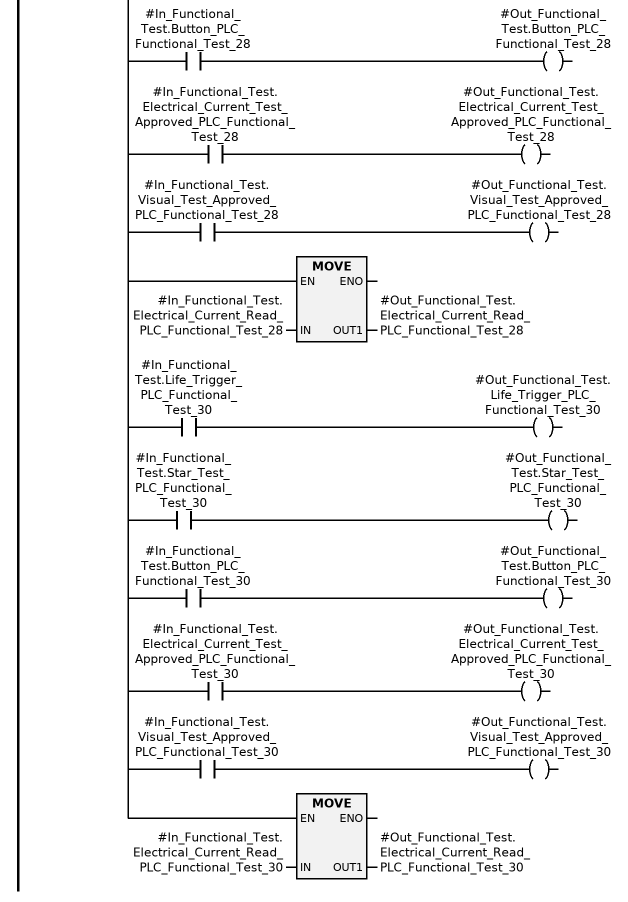
   RUNG wire#powerrail
      { S7_Templates := "SrcType := SInt" } EQ_Contact(in1 := #Test_Station, in2 := 14)
      wire#w1
      Contact( #Life_Trigger )
      Coil( #Out_Functional_Test.Life_Trigger_PLC_Functional_Test_14 )
   END_RUNG
   RUNG wire#w1
      Contact( #Star_Test )
      Coil( #Out_Functional_Test.Star_Test_PLC_Functional_Test_14 )
   END_RUNG
   RUNG wire#w1
      Contact( #Button_Start_Approve )
      Coil( #Out_Functional_Test.Button_PLC_Functional_Test_14 )
   END_RUNG
   RUNG wire#w1
      Contact( #Electrical_Current_Test_Approved )
      Coil( #Out_Functional_Test.Electrical_Current_Test_Approved_PLC_Functional_Test_14 )
   END_RUNG
   RUNG wire#w1
      Contact( #Visual_Test_Approved )
      Coil( #Out_Functional_Test.Visual_Test_Approved_PLC_Functional_Test_14 )
   END_RUNG
   RUNG wire#w1
      Contact( #In_Test_Parameters.Reset_PLC_Functional_Test_14 )
      Coil( #Reset_Functional_Test )
   END_RUNG
   RUNG wire#w1
      Move(in := #Electrical_Current_Read, out1 => #Out_Functional_Test.Electrical_Current_Read_PLC_Functional_Test_14)
   END_RUNG
   RUNG wire#w1
      Contact( #In_Functional_Test.Life_Trigger_PLC_Functional_Test_16 )
      Coil( #Out_Functional_Test.Life_Trigger_PLC_Functional_Test_16 )
   END_RUNG
   RUNG wire#w1
      Contact( #In_Functional_Test.Star_Test_PLC_Functional_Test_16 )
      Coil( #Out_Functional_Test.Star_Test_PLC_Functional_Test_16 )
   END_RUNG
   RUNG wire#w1
      Contact( #In_Functional_Test.Button_PLC_Functional_Test_16 )
      Coil( #Out_Functional_Test.Button_PLC_Functional_Test_16 )
   END_RUNG
   RUNG wire#w1
      Contact( #In_Functional_Test.Electrical_Current_Test_Approved_PLC_Functional_Test_16 )
      Coil( #Out_Functional_Test.Electrical_Current_Test_Approved_PLC_Functional_Test_16 )
   END_RUNG
   RUNG wire#w1
      Contact( #In_Functional_Test.Visual_Test_Approved_PLC_Functional_Test_16 )
      Coil( #Out_Functional_Test.Visual_Test_Approved_PLC_Functional_Test_16 )
   END_RUNG
   RUNG wire#w1
      Move(in := #In_Functional_Test.Electrical_Current_Read_PLC_Functional_Test_16, out1 => #Out_Functional_Test.Electrical_Current_Read_PLC_Functional_Test_16)
   END_RUNG
   RUNG wire#w1
      Contact( #In_Functional_Test.Life_Trigger_PLC_Functional_Test_18 )
      Coil( #Out_Functional_Test.Life_Trigger_PLC_Functional_Test_18 )
   END_RUNG
   RUNG wire#w1
      Contact( #In_Functional_Test.Star_Test_PLC_Functional_Test_18 )
      Coil( #Out_Functional_Test.Star_Test_PLC_Functional_Test_18 )
   END_RUNG
   RUNG wire#w1
      Contact( #In_Functional_Test.Button_PLC_Functional_Test_18 )
      Coil( #Out_Functional_Test.Button_PLC_Functional_Test_18 )
   END_RUNG
   RUNG wire#w1
      Contact( #In_Functional_Test.Electrical_Current_Test_Approved_PLC_Functional_Test_18 )
      Coil( #Out_Functional_Test.Electrical_Current_Test_Approved_PLC_Functional_Test_18 )
   END_RUNG
   RUNG wire#w1
      Contact( #In_Functional_Test.Visual_Test_Approved_PLC_Functional_Test_18 )
      Coil( #Out_Functional_Test.Visual_Test_Approved_PLC_Functional_Test_18 )
   END_RUNG
   RUNG wire#w1
      Move(in := #In_Functional_Test.Electrical_Current_Read_PLC_Functional_Test_18, out1 => #Out_Functional_Test.Electrical_Current_Read_PLC_Functional_Test_18)
   END_RUNG
   RUNG wire#w1
      Contact( #In_Functional_Test.Life_Trigger_PLC_Functional_Test_20 )
      Coil( #Out_Functional_Test.Life_Trigger_PLC_Functional_Test_20 )
   END_RUNG
   RUNG wire#w1
      Contact( #In_Functional_Test.Star_Test_PLC_Functional_Test_20 )
      Coil( #Out_Functional_Test.Star_Test_PLC_Functional_Test_20 )
   END_RUNG
   RUNG wire#w1
      Contact( #In_Functional_Test.Button_PLC_Functional_Test_20 )
      Coil( #Out_Functional_Test.Button_PLC_Functional_Test_20 )
   END_RUNG
   RUNG wire#w1
      Contact( #In_Functional_Test.Electrical_Current_Test_Approved_PLC_Functional_Test_20 )
      Coil( #Out_Functional_Test.Electrical_Current_Test_Approved_PLC_Functional_Test_20 )
   END_RUNG
   RUNG wire#w1
      Contact( #In_Functional_Test.Visual_Test_Approved_PLC_Functional_Test_20 )
      Coil( #Out_Functional_Test.Visual_Test_Approved_PLC_Functional_Test_20 )
   END_RUNG
   RUNG wire#w1
      Move(in := #In_Functional_Test.Electrical_Current_Read_PLC_Functional_Test_20, out1 => #Out_Functional_Test.Electrical_Current_Read_PLC_Functional_Test_20)
   END_RUNG
   RUNG wire#w1
      Contact( #In_Functional_Test.Life_Trigger_PLC_Functional_Test_22 )
      Coil( #Out_Functional_Test.Life_Trigger_PLC_Functional_Test_22 )
   END_RUNG
   RUNG wire#w1
      Contact( #In_Functional_Test.Star_Test_PLC_Functional_Test_22 )
      Coil( #Out_Functional_Test.Star_Test_PLC_Functional_Test_22 )
   END_RUNG
   RUNG wire#w1
      Contact( #In_Functional_Test.Button_PLC_Functional_Test_22 )
      Coil( #Out_Functional_Test.Button_PLC_Functional_Test_22 )
   END_RUNG
   RUNG wire#w1
      Contact( #In_Functional_Test.Electrical_Current_Test_Approved_PLC_Functional_Test_22 )
      Coil( #Out_Functional_Test.Electrical_Current_Test_Approved_PLC_Functional_Test_22 )
   END_RUNG
   RUNG wire#w1
      Contact( #In_Functional_Test.Visual_Test_Approved_PLC_Functional_Test_22 )
      Coil( #Out_Functional_Test.Visual_Test_Approved_PLC_Functional_Test_22 )
   END_RUNG
   RUNG wire#w1
      Move(in := #In_Functional_Test.Electrical_Current_Read_PLC_Functional_Test_22, out1 => #Out_Functional_Test.Electrical_Current_Read_PLC_Functional_Test_22)
   END_RUNG
   RUNG wire#w1
      Contact( #In_Functional_Test.Life_Trigger_PLC_Functional_Test_24 )
      Coil( #Out_Functional_Test.Life_Trigger_PLC_Functional_Test_24 )
   END_RUNG
   RUNG wire#w1
      Contact( #In_Functional_Test.Star_Test_PLC_Functional_Test_24 )
      Coil( #Out_Functional_Test.Star_Test_PLC_Functional_Test_24 )
   END_RUNG
   RUNG wire#w1
      Contact( #In_Functional_Test.Button_PLC_Functional_Test_24 )
      Coil( #Out_Functional_Test.Button_PLC_Functional_Test_24 )
   END_RUNG
   RUNG wire#w1
      Contact( #In_Functional_Test.Electrical_Current_Test_Approved_PLC_Functional_Test_24 )
      Coil( #Out_Functional_Test.Electrical_Current_Test_Approved_PLC_Functional_Test_24 )
   END_RUNG
   RUNG wire#w1
      Contact( #In_Functional_Test.Visual_Test_Approved_PLC_Functional_Test_24 )
      Coil( #Out_Functional_Test.Visual_Test_Approved_PLC_Functional_Test_24 )
   END_RUNG
   RUNG wire#w1
      Move(in := #In_Functional_Test.Electrical_Current_Read_PLC_Functional_Test_24, out1 => #Out_Functional_Test.Electrical_Current_Read_PLC_Functional_Test_24)
   END_RUNG
   RUNG wire#w1
      Contact( #In_Functional_Test.Life_Trigger_PLC_Functional_Test_26 )
      Coil( #Out_Functional_Test.Life_Trigger_PLC_Functional_Test_26 )
   END_RUNG
   RUNG wire#w1
      Contact( #In_Functional_Test.Star_Test_PLC_Functional_Test_26 )
      Coil( #Out_Functional_Test.Star_Test_PLC_Functional_Test_26 )
   END_RUNG
   RUNG wire#w1
      Contact( #In_Functional_Test.Button_PLC_Functional_Test_26 )
      Coil( #Out_Functional_Test.Button_PLC_Functional_Test_26 )
   END_RUNG
   RUNG wire#w1
      Contact( #In_Functional_Test.Electrical_Current_Test_Approved_PLC_Functional_Test_26 )
      Coil( #Out_Functional_Test.Electrical_Current_Test_Approved_PLC_Functional_Test_26 )
   END_RUNG
   RUNG wire#w1
      Contact( #In_Functional_Test.Visual_Test_Approved_PLC_Functional_Test_26 )
      Coil( #Out_Functional_Test.Visual_Test_Approved_PLC_Functional_Test_26 )
   END_RUNG
   RUNG wire#w1
      Move(in := #In_Functional_Test.Electrical_Current_Read_PLC_Functional_Test_26, out1 => #Out_Functional_Test.Electrical_Current_Read_PLC_Functional_Test_26)
   END_RUNG
   RUNG wire#w1
      Contact( #In_Functional_Test.Life_Trigger_PLC_Functional_Test_28 )
      Coil( #Out_Functional_Test.Life_Trigger_PLC_Functional_Test_28 )
   END_RUNG
   RUNG wire#w1
      Contact( #In_Functional_Test.Star_Test_PLC_Functional_Test_28 )
      Coil( #Out_Functional_Test.Star_Test_PLC_Functional_Test_28 )
   END_RUNG
   RUNG wire#w1
      Contact( #In_Functional_Test.Button_PLC_Functional_Test_28 )
      Coil( #Out_Functional_Test.Button_PLC_Functional_Test_28 )
   END_RUNG
   RUNG wire#w1
      Contact( #In_Functional_Test.Electrical_Current_Test_Approved_PLC_Functional_Test_28 )
      Coil( #Out_Functional_Test.Electrical_Current_Test_Approved_PLC_Functional_Test_28 )
   END_RUNG
   RUNG wire#w1
      Contact( #In_Functional_Test.Visual_Test_Approved_PLC_Functional_Test_28 )
      Coil( #Out_Functional_Test.Visual_Test_Approved_PLC_Functional_Test_28 )
   END_RUNG
   RUNG wire#w1
      Move(in := #In_Functional_Test.Electrical_Current_Read_PLC_Functional_Test_28, out1 => #Out_Functional_Test.Electrical_Current_Read_PLC_Functional_Test_28)
   END_RUNG
   RUNG wire#w1
      Contact( #In_Functional_Test.Life_Trigger_PLC_Functional_Test_30 )
      Coil( #Out_Functional_Test.Life_Trigger_PLC_Functional_Test_30 )
   END_RUNG
   RUNG wire#w1
      Contact( #In_Functional_Test.Star_Test_PLC_Functional_Test_30 )
      Coil( #Out_Functional_Test.Star_Test_PLC_Functional_Test_30 )
   END_RUNG
   RUNG wire#w1
      Contact( #In_Functional_Test.Button_PLC_Functional_Test_30 )
      Coil( #Out_Functional_Test.Button_PLC_Functional_Test_30 )
   END_RUNG
   RUNG wire#w1
      Contact( #In_Functional_Test.Electrical_Current_Test_Approved_PLC_Functional_Test_30 )
      Coil( #Out_Functional_Test.Electrical_Current_Test_Approved_PLC_Functional_Test_30 )
   END_RUNG
   RUNG wire#w1
      Contact( #In_Functional_Test.Visual_Test_Approved_PLC_Functional_Test_30 )
      Coil( #Out_Functional_Test.Visual_Test_Approved_PLC_Functional_Test_30 )
   END_RUNG
   RUNG wire#w1
      Move(in := #In_Functional_Test.Electrical_Current_Read_PLC_Functional_Test_30, out1 => #Out_Functional_Test.Electrical_Current_Read_PLC_Functional_Test_30)
   END_RUNG
   // the same network as SCL:
   #_w1 := #Test_Station = 14;
   #Out_Functional_Test.Life_Trigger_PLC_Functional_Test_14 := #_w1 AND #Life_Trigger;
   #Out_Functional_Test.Star_Test_PLC_Functional_Test_14 := #_w1 AND #Star_Test;
   #Out_Functional_Test.Button_PLC_Functional_Test_14 := #_w1 AND #Button_Start_Approve;
   #Out_Functional_Test.Electrical_Current_Test_Approved_PLC_Functional_Test_14 := #_w1 AND #Electrical_Current_Test_Approved;
   #Out_Functional_Test.Visual_Test_Approved_PLC_Functional_Test_14 := #_w1 AND #Visual_Test_Approved;
   #Reset_Functional_Test := #_w1 AND #In_Test_Parameters.Reset_PLC_Functional_Test_14;
   IF #_w1 THEN
       #Out_Functional_Test.Electrical_Current_Read_PLC_Functional_Test_14 := #Electrical_Current_Read;
   END_IF;
   #Out_Functional_Test.Life_Trigger_PLC_Functional_Test_16 := #_w1 AND #In_Functional_Test.Life_Trigger_PLC_Functional_Test_16;
   #Out_Functional_Test.Star_Test_PLC_Functional_Test_16 := #_w1 AND #In_Functional_Test.Star_Test_PLC_Functional_Test_16;
   #Out_Functional_Test.Button_PLC_Functional_Test_16 := #_w1 AND #In_Functional_Test.Button_PLC_Functional_Test_16;
   #Out_Functional_Test.Electrical_Current_Test_Approved_PLC_Functional_Test_16 := #_w1 AND #In_Functional_Test.Electrical_Current_Test_Approved_PLC_Functional_Test_16;
   #Out_Functional_Test.Visual_Test_Approved_PLC_Functional_Test_16 := #_w1 AND #In_Functional_Test.Visual_Test_Approved_PLC_Functional_Test_16;
   IF #_w1 THEN
       #Out_Functional_Test.Electrical_Current_Read_PLC_Functional_Test_16 := #In_Functional_Test.Electrical_Current_Read_PLC_Functional_Test_16;
   END_IF;
   #Out_Functional_Test.Life_Trigger_PLC_Functional_Test_18 := #_w1 AND #In_Functional_Test.Life_Trigger_PLC_Functional_Test_18;
   #Out_Functional_Test.Star_Test_PLC_Functional_Test_18 := #_w1 AND #In_Functional_Test.Star_Test_PLC_Functional_Test_18;
   #Out_Functional_Test.Button_PLC_Functional_Test_18 := #_w1 AND #In_Functional_Test.Button_PLC_Functional_Test_18;
   #Out_Functional_Test.Electrical_Current_Test_Approved_PLC_Functional_Test_18 := #_w1 AND #In_Functional_Test.Electrical_Current_Test_Approved_PLC_Functional_Test_18;
   #Out_Functional_Test.Visual_Test_Approved_PLC_Functional_Test_18 := #_w1 AND #In_Functional_Test.Visual_Test_Approved_PLC_Functional_Test_18;
   IF #_w1 THEN
       #Out_Functional_Test.Electrical_Current_Read_PLC_Functional_Test_18 := #In_Functional_Test.Electrical_Current_Read_PLC_Functional_Test_18;
   END_IF;
   #Out_Functional_Test.Life_Trigger_PLC_Functional_Test_20 := #_w1 AND #In_Functional_Test.Life_Trigger_PLC_Functional_Test_20;
   #Out_Functional_Test.Star_Test_PLC_Functional_Test_20 := #_w1 AND #In_Functional_Test.Star_Test_PLC_Functional_Test_20;
   #Out_Functional_Test.Button_PLC_Functional_Test_20 := #_w1 AND #In_Functional_Test.Button_PLC_Functional_Test_20;
   #Out_Functional_Test.Electrical_Current_Test_Approved_PLC_Functional_Test_20 := #_w1 AND #In_Functional_Test.Electrical_Current_Test_Approved_PLC_Functional_Test_20;
   #Out_Functional_Test.Visual_Test_Approved_PLC_Functional_Test_20 := #_w1 AND #In_Functional_Test.Visual_Test_Approved_PLC_Functional_Test_20;
   IF #_w1 THEN
       #Out_Functional_Test.Electrical_Current_Read_PLC_Functional_Test_20 := #In_Functional_Test.Electrical_Current_Read_PLC_Functional_Test_20;
   END_IF;
   #Out_Functional_Test.Life_Trigger_PLC_Functional_Test_22 := #_w1 AND #In_Functional_Test.Life_Trigger_PLC_Functional_Test_22;
   #Out_Functional_Test.Star_Test_PLC_Functional_Test_22 := #_w1 AND #In_Functional_Test.Star_Test_PLC_Functional_Test_22;
   #Out_Functional_Test.Button_PLC_Functional_Test_22 := #_w1 AND #In_Functional_Test.Button_PLC_Functional_Test_22;
   #Out_Functional_Test.Electrical_Current_Test_Approved_PLC_Functional_Test_22 := #_w1 AND #In_Functional_Test.Electrical_Current_Test_Approved_PLC_Functional_Test_22;
   #Out_Functional_Test.Visual_Test_Approved_PLC_Functional_Test_22 := #_w1 AND #In_Functional_Test.Visual_Test_Approved_PLC_Functional_Test_22;
   IF #_w1 THEN
       #Out_Functional_Test.Electrical_Current_Read_PLC_Functional_Test_22 := #In_Functional_Test.Electrical_Current_Read_PLC_Functional_Test_22;
   END_IF;
   #Out_Functional_Test.Life_Trigger_PLC_Functional_Test_24 := #_w1 AND #In_Functional_Test.Life_Trigger_PLC_Functional_Test_24;
   #Out_Functional_Test.Star_Test_PLC_Functional_Test_24 := #_w1 AND #In_Functional_Test.Star_Test_PLC_Functional_Test_24;
   #Out_Functional_Test.Button_PLC_Functional_Test_24 := #_w1 AND #In_Functional_Test.Button_PLC_Functional_Test_24;
   #Out_Functional_Test.Electrical_Current_Test_Approved_PLC_Functional_Test_24 := #_w1 AND #In_Functional_Test.Electrical_Current_Test_Approved_PLC_Functional_Test_24;
   #Out_Functional_Test.Visual_Test_Approved_PLC_Functional_Test_24 := #_w1 AND #In_Functional_Test.Visual_Test_Approved_PLC_Functional_Test_24;
   IF #_w1 THEN
       #Out_Functional_Test.Electrical_Current_Read_PLC_Functional_Test_24 := #In_Functional_Test.Electrical_Current_Read_PLC_Functional_Test_24;
   END_IF;
   #Out_Functional_Test.Life_Trigger_PLC_Functional_Test_26 := #_w1 AND #In_Functional_Test.Life_Trigger_PLC_Functional_Test_26;
   #Out_Functional_Test.Star_Test_PLC_Functional_Test_26 := #_w1 AND #In_Functional_Test.Star_Test_PLC_Functional_Test_26;
   #Out_Functional_Test.Button_PLC_Functional_Test_26 := #_w1 AND #In_Functional_Test.Button_PLC_Functional_Test_26;
   #Out_Functional_Test.Electrical_Current_Test_Approved_PLC_Functional_Test_26 := #_w1 AND #In_Functional_Test.Electrical_Current_Test_Approved_PLC_Functional_Test_26;
   #Out_Functional_Test.Visual_Test_Approved_PLC_Functional_Test_26 := #_w1 AND #In_Functional_Test.Visual_Test_Approved_PLC_Functional_Test_26;
   IF #_w1 THEN
       #Out_Functional_Test.Electrical_Current_Read_PLC_Functional_Test_26 := #In_Functional_Test.Electrical_Current_Read_PLC_Functional_Test_26;
   END_IF;
   #Out_Functional_Test.Life_Trigger_PLC_Functional_Test_28 := #_w1 AND #In_Functional_Test.Life_Trigger_PLC_Functional_Test_28;
   #Out_Functional_Test.Star_Test_PLC_Functional_Test_28 := #_w1 AND #In_Functional_Test.Star_Test_PLC_Functional_Test_28;
   #Out_Functional_Test.Button_PLC_Functional_Test_28 := #_w1 AND #In_Functional_Test.Button_PLC_Functional_Test_28;
   #Out_Functional_Test.Electrical_Current_Test_Approved_PLC_Functional_Test_28 := #_w1 AND #In_Functional_Test.Electrical_Current_Test_Approved_PLC_Functional_Test_28;
   #Out_Functional_Test.Visual_Test_Approved_PLC_Functional_Test_28 := #_w1 AND #In_Functional_Test.Visual_Test_Approved_PLC_Functional_Test_28;
   IF #_w1 THEN
       #Out_Functional_Test.Electrical_Current_Read_PLC_Functional_Test_28 := #In_Functional_Test.Electrical_Current_Read_PLC_Functional_Test_28;
   END_IF;
   #Out_Functional_Test.Life_Trigger_PLC_Functional_Test_30 := #_w1 AND #In_Functional_Test.Life_Trigger_PLC_Functional_Test_30;
   #Out_Functional_Test.Star_Test_PLC_Functional_Test_30 := #_w1 AND #In_Functional_Test.Star_Test_PLC_Functional_Test_30;
   #Out_Functional_Test.Button_PLC_Functional_Test_30 := #_w1 AND #In_Functional_Test.Button_PLC_Functional_Test_30;
   #Out_Functional_Test.Electrical_Current_Test_Approved_PLC_Functional_Test_30 := #_w1 AND #In_Functional_Test.Electrical_Current_Test_Approved_PLC_Functional_Test_30;
   #Out_Functional_Test.Visual_Test_Approved_PLC_Functional_Test_30 := #_w1 AND #In_Functional_Test.Visual_Test_Approved_PLC_Functional_Test_30;
   IF #_w1 THEN
       #Out_Functional_Test.Electrical_Current_Read_PLC_Functional_Test_30 := #In_Functional_Test.Electrical_Current_Read_PLC_Functional_Test_30;
   END_IF;
END_REGION

REGION Network 9: Functional Test Station 16
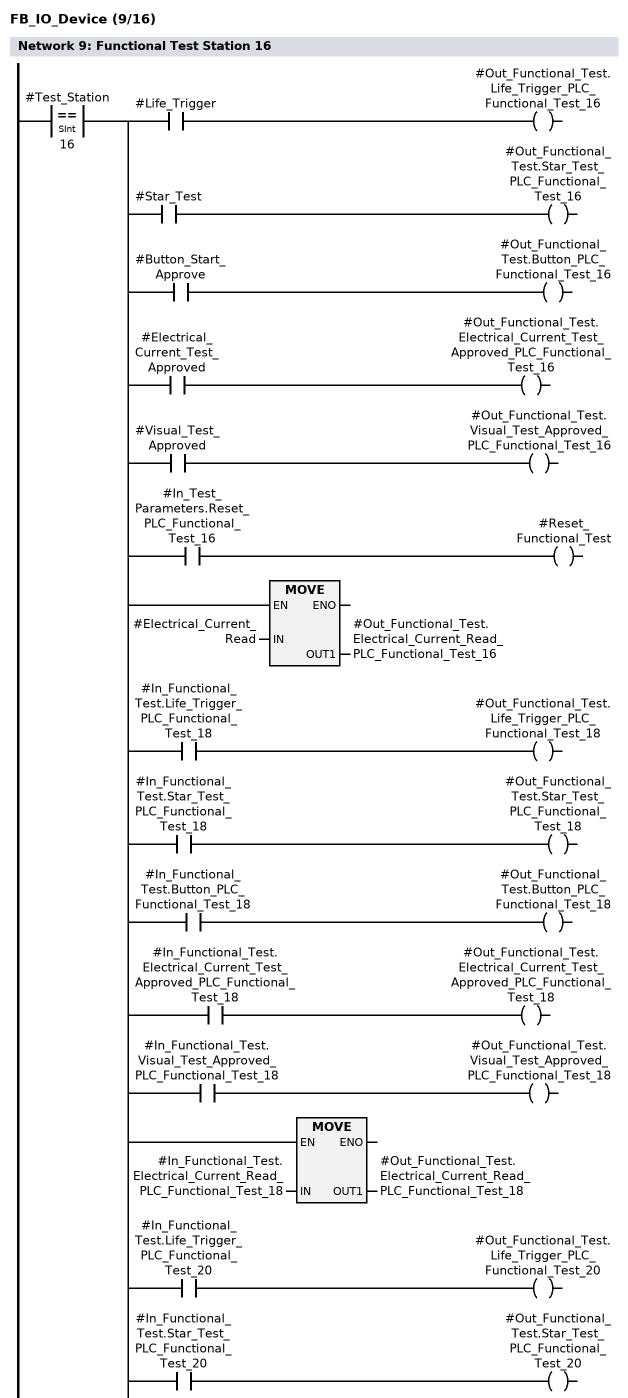
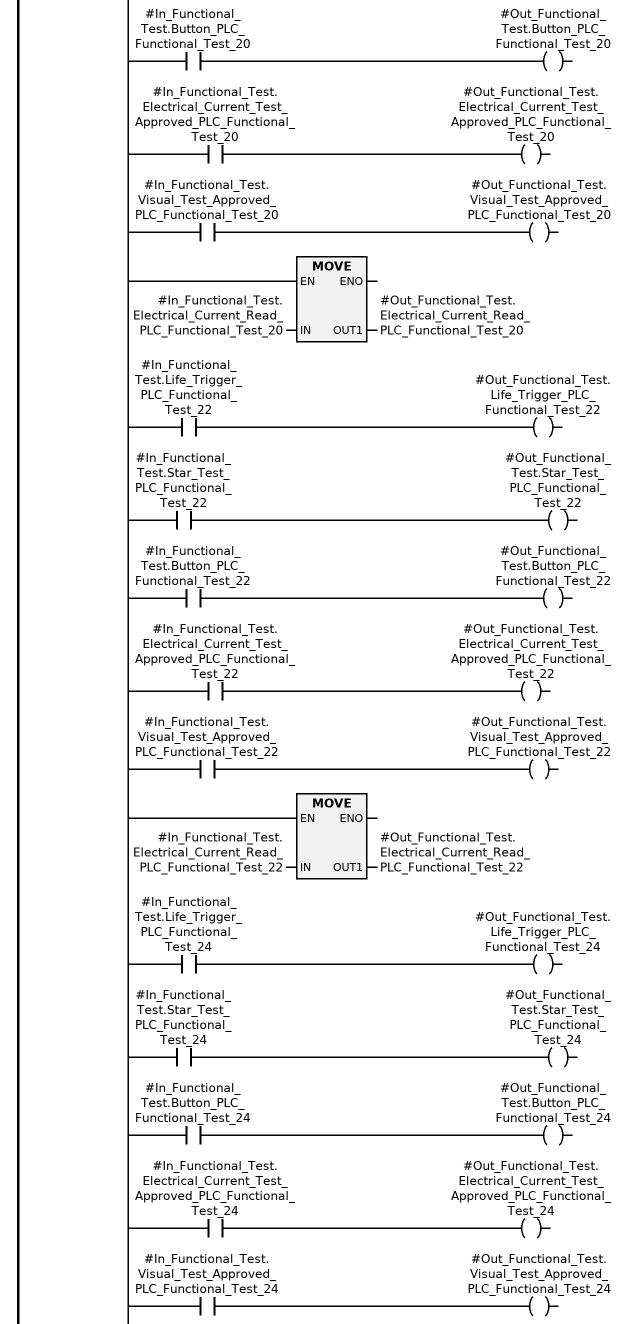
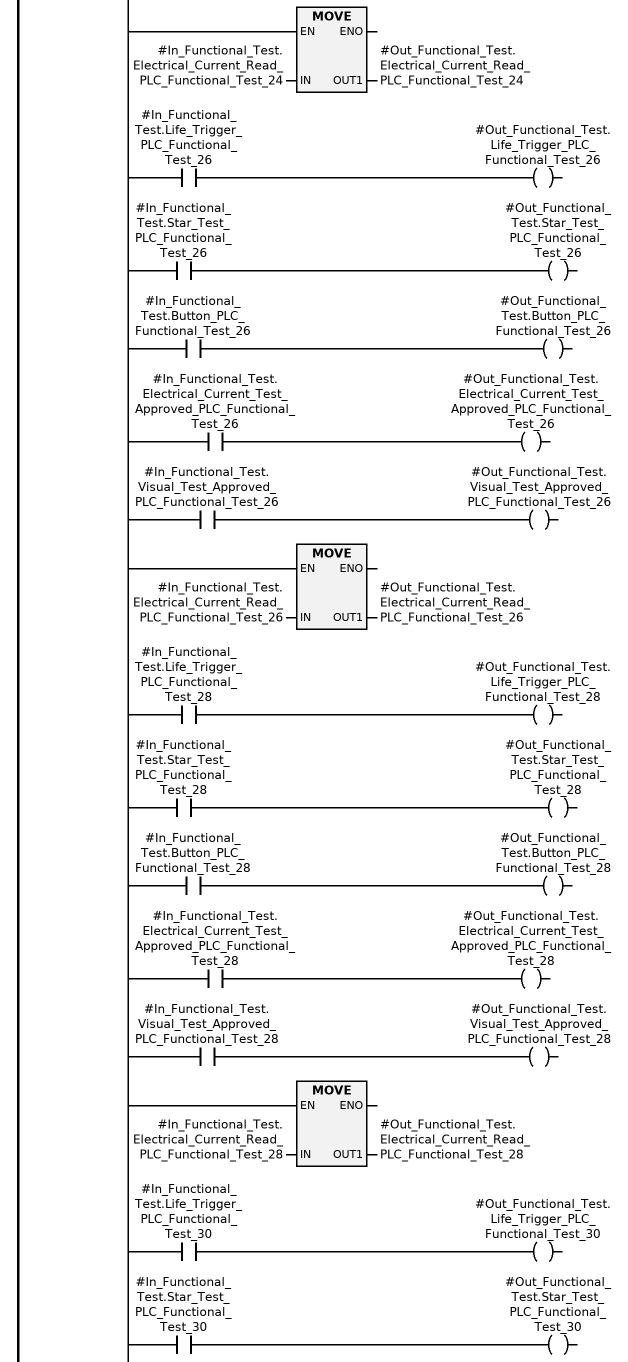
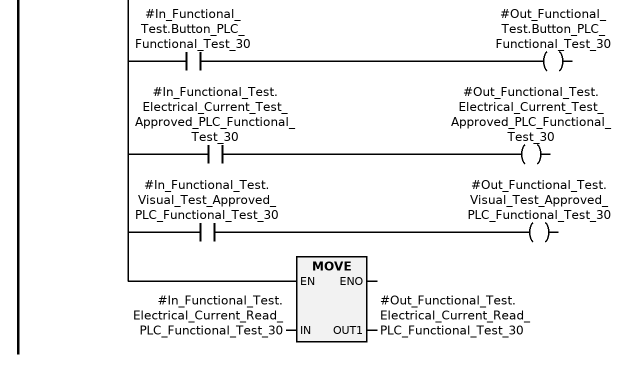
   RUNG wire#powerrail
      { S7_Templates := "SrcType := SInt" } EQ_Contact(in1 := #Test_Station, in2 := 16)
      wire#w1
      Contact( #Life_Trigger )
      Coil( #Out_Functional_Test.Life_Trigger_PLC_Functional_Test_16 )
   END_RUNG
   RUNG wire#w1
      Contact( #Star_Test )
      Coil( #Out_Functional_Test.Star_Test_PLC_Functional_Test_16 )
   END_RUNG
   RUNG wire#w1
      Contact( #Button_Start_Approve )
      Coil( #Out_Functional_Test.Button_PLC_Functional_Test_16 )
   END_RUNG
   RUNG wire#w1
      Contact( #Electrical_Current_Test_Approved )
      Coil( #Out_Functional_Test.Electrical_Current_Test_Approved_PLC_Functional_Test_16 )
   END_RUNG
   RUNG wire#w1
      Contact( #Visual_Test_Approved )
      Coil( #Out_Functional_Test.Visual_Test_Approved_PLC_Functional_Test_16 )
   END_RUNG
   RUNG wire#w1
      Contact( #In_Test_Parameters.Reset_PLC_Functional_Test_16 )
      Coil( #Reset_Functional_Test )
   END_RUNG
   RUNG wire#w1
      Move(in := #Electrical_Current_Read, out1 => #Out_Functional_Test.Electrical_Current_Read_PLC_Functional_Test_16)
   END_RUNG
   RUNG wire#w1
      Contact( #In_Functional_Test.Life_Trigger_PLC_Functional_Test_18 )
      Coil( #Out_Functional_Test.Life_Trigger_PLC_Functional_Test_18 )
   END_RUNG
   RUNG wire#w1
      Contact( #In_Functional_Test.Star_Test_PLC_Functional_Test_18 )
      Coil( #Out_Functional_Test.Star_Test_PLC_Functional_Test_18 )
   END_RUNG
   RUNG wire#w1
      Contact( #In_Functional_Test.Button_PLC_Functional_Test_18 )
      Coil( #Out_Functional_Test.Button_PLC_Functional_Test_18 )
   END_RUNG
   RUNG wire#w1
      Contact( #In_Functional_Test.Electrical_Current_Test_Approved_PLC_Functional_Test_18 )
      Coil( #Out_Functional_Test.Electrical_Current_Test_Approved_PLC_Functional_Test_18 )
   END_RUNG
   RUNG wire#w1
      Contact( #In_Functional_Test.Visual_Test_Approved_PLC_Functional_Test_18 )
      Coil( #Out_Functional_Test.Visual_Test_Approved_PLC_Functional_Test_18 )
   END_RUNG
   RUNG wire#w1
      Move(in := #In_Functional_Test.Electrical_Current_Read_PLC_Functional_Test_18, out1 => #Out_Functional_Test.Electrical_Current_Read_PLC_Functional_Test_18)
   END_RUNG
   RUNG wire#w1
      Contact( #In_Functional_Test.Life_Trigger_PLC_Functional_Test_20 )
      Coil( #Out_Functional_Test.Life_Trigger_PLC_Functional_Test_20 )
   END_RUNG
   RUNG wire#w1
      Contact( #In_Functional_Test.Star_Test_PLC_Functional_Test_20 )
      Coil( #Out_Functional_Test.Star_Test_PLC_Functional_Test_20 )
   END_RUNG
   RUNG wire#w1
      Contact( #In_Functional_Test.Button_PLC_Functional_Test_20 )
      Coil( #Out_Functional_Test.Button_PLC_Functional_Test_20 )
   END_RUNG
   RUNG wire#w1
      Contact( #In_Functional_Test.Electrical_Current_Test_Approved_PLC_Functional_Test_20 )
      Coil( #Out_Functional_Test.Electrical_Current_Test_Approved_PLC_Functional_Test_20 )
   END_RUNG
   RUNG wire#w1
      Contact( #In_Functional_Test.Visual_Test_Approved_PLC_Functional_Test_20 )
      Coil( #Out_Functional_Test.Visual_Test_Approved_PLC_Functional_Test_20 )
   END_RUNG
   RUNG wire#w1
      Move(in := #In_Functional_Test.Electrical_Current_Read_PLC_Functional_Test_20, out1 => #Out_Functional_Test.Electrical_Current_Read_PLC_Functional_Test_20)
   END_RUNG
   RUNG wire#w1
      Contact( #In_Functional_Test.Life_Trigger_PLC_Functional_Test_22 )
      Coil( #Out_Functional_Test.Life_Trigger_PLC_Functional_Test_22 )
   END_RUNG
   RUNG wire#w1
      Contact( #In_Functional_Test.Star_Test_PLC_Functional_Test_22 )
      Coil( #Out_Functional_Test.Star_Test_PLC_Functional_Test_22 )
   END_RUNG
   RUNG wire#w1
      Contact( #In_Functional_Test.Button_PLC_Functional_Test_22 )
      Coil( #Out_Functional_Test.Button_PLC_Functional_Test_22 )
   END_RUNG
   RUNG wire#w1
      Contact( #In_Functional_Test.Electrical_Current_Test_Approved_PLC_Functional_Test_22 )
      Coil( #Out_Functional_Test.Electrical_Current_Test_Approved_PLC_Functional_Test_22 )
   END_RUNG
   RUNG wire#w1
      Contact( #In_Functional_Test.Visual_Test_Approved_PLC_Functional_Test_22 )
      Coil( #Out_Functional_Test.Visual_Test_Approved_PLC_Functional_Test_22 )
   END_RUNG
   RUNG wire#w1
      Move(in := #In_Functional_Test.Electrical_Current_Read_PLC_Functional_Test_22, out1 => #Out_Functional_Test.Electrical_Current_Read_PLC_Functional_Test_22)
   END_RUNG
   RUNG wire#w1
      Contact( #In_Functional_Test.Life_Trigger_PLC_Functional_Test_24 )
      Coil( #Out_Functional_Test.Life_Trigger_PLC_Functional_Test_24 )
   END_RUNG
   RUNG wire#w1
      Contact( #In_Functional_Test.Star_Test_PLC_Functional_Test_24 )
      Coil( #Out_Functional_Test.Star_Test_PLC_Functional_Test_24 )
   END_RUNG
   RUNG wire#w1
      Contact( #In_Functional_Test.Button_PLC_Functional_Test_24 )
      Coil( #Out_Functional_Test.Button_PLC_Functional_Test_24 )
   END_RUNG
   RUNG wire#w1
      Contact( #In_Functional_Test.Electrical_Current_Test_Approved_PLC_Functional_Test_24 )
      Coil( #Out_Functional_Test.Electrical_Current_Test_Approved_PLC_Functional_Test_24 )
   END_RUNG
   RUNG wire#w1
      Contact( #In_Functional_Test.Visual_Test_Approved_PLC_Functional_Test_24 )
      Coil( #Out_Functional_Test.Visual_Test_Approved_PLC_Functional_Test_24 )
   END_RUNG
   RUNG wire#w1
      Move(in := #In_Functional_Test.Electrical_Current_Read_PLC_Functional_Test_24, out1 => #Out_Functional_Test.Electrical_Current_Read_PLC_Functional_Test_24)
   END_RUNG
   RUNG wire#w1
      Contact( #In_Functional_Test.Life_Trigger_PLC_Functional_Test_26 )
      Coil( #Out_Functional_Test.Life_Trigger_PLC_Functional_Test_26 )
   END_RUNG
   RUNG wire#w1
      Contact( #In_Functional_Test.Star_Test_PLC_Functional_Test_26 )
      Coil( #Out_Functional_Test.Star_Test_PLC_Functional_Test_26 )
   END_RUNG
   RUNG wire#w1
      Contact( #In_Functional_Test.Button_PLC_Functional_Test_26 )
      Coil( #Out_Functional_Test.Button_PLC_Functional_Test_26 )
   END_RUNG
   RUNG wire#w1
      Contact( #In_Functional_Test.Electrical_Current_Test_Approved_PLC_Functional_Test_26 )
      Coil( #Out_Functional_Test.Electrical_Current_Test_Approved_PLC_Functional_Test_26 )
   END_RUNG
   RUNG wire#w1
      Contact( #In_Functional_Test.Visual_Test_Approved_PLC_Functional_Test_26 )
      Coil( #Out_Functional_Test.Visual_Test_Approved_PLC_Functional_Test_26 )
   END_RUNG
   RUNG wire#w1
      Move(in := #In_Functional_Test.Electrical_Current_Read_PLC_Functional_Test_26, out1 => #Out_Functional_Test.Electrical_Current_Read_PLC_Functional_Test_26)
   END_RUNG
   RUNG wire#w1
      Contact( #In_Functional_Test.Life_Trigger_PLC_Functional_Test_28 )
      Coil( #Out_Functional_Test.Life_Trigger_PLC_Functional_Test_28 )
   END_RUNG
   RUNG wire#w1
      Contact( #In_Functional_Test.Star_Test_PLC_Functional_Test_28 )
      Coil( #Out_Functional_Test.Star_Test_PLC_Functional_Test_28 )
   END_RUNG
   RUNG wire#w1
      Contact( #In_Functional_Test.Button_PLC_Functional_Test_28 )
      Coil( #Out_Functional_Test.Button_PLC_Functional_Test_28 )
   END_RUNG
   RUNG wire#w1
      Contact( #In_Functional_Test.Electrical_Current_Test_Approved_PLC_Functional_Test_28 )
      Coil( #Out_Functional_Test.Electrical_Current_Test_Approved_PLC_Functional_Test_28 )
   END_RUNG
   RUNG wire#w1
      Contact( #In_Functional_Test.Visual_Test_Approved_PLC_Functional_Test_28 )
      Coil( #Out_Functional_Test.Visual_Test_Approved_PLC_Functional_Test_28 )
   END_RUNG
   RUNG wire#w1
      Move(in := #In_Functional_Test.Electrical_Current_Read_PLC_Functional_Test_28, out1 => #Out_Functional_Test.Electrical_Current_Read_PLC_Functional_Test_28)
   END_RUNG
   RUNG wire#w1
      Contact( #In_Functional_Test.Life_Trigger_PLC_Functional_Test_30 )
      Coil( #Out_Functional_Test.Life_Trigger_PLC_Functional_Test_30 )
   END_RUNG
   RUNG wire#w1
      Contact( #In_Functional_Test.Star_Test_PLC_Functional_Test_30 )
      Coil( #Out_Functional_Test.Star_Test_PLC_Functional_Test_30 )
   END_RUNG
   RUNG wire#w1
      Contact( #In_Functional_Test.Button_PLC_Functional_Test_30 )
      Coil( #Out_Functional_Test.Button_PLC_Functional_Test_30 )
   END_RUNG
   RUNG wire#w1
      Contact( #In_Functional_Test.Electrical_Current_Test_Approved_PLC_Functional_Test_30 )
      Coil( #Out_Functional_Test.Electrical_Current_Test_Approved_PLC_Functional_Test_30 )
   END_RUNG
   RUNG wire#w1
      Contact( #In_Functional_Test.Visual_Test_Approved_PLC_Functional_Test_30 )
      Coil( #Out_Functional_Test.Visual_Test_Approved_PLC_Functional_Test_30 )
   END_RUNG
   RUNG wire#w1
      Move(in := #In_Functional_Test.Electrical_Current_Read_PLC_Functional_Test_30, out1 => #Out_Functional_Test.Electrical_Current_Read_PLC_Functional_Test_30)
   END_RUNG
   // the same network as SCL:
   #_w1 := #Test_Station = 16;
   #Out_Functional_Test.Life_Trigger_PLC_Functional_Test_16 := #_w1 AND #Life_Trigger;
   #Out_Functional_Test.Star_Test_PLC_Functional_Test_16 := #_w1 AND #Star_Test;
   #Out_Functional_Test.Button_PLC_Functional_Test_16 := #_w1 AND #Button_Start_Approve;
   #Out_Functional_Test.Electrical_Current_Test_Approved_PLC_Functional_Test_16 := #_w1 AND #Electrical_Current_Test_Approved;
   #Out_Functional_Test.Visual_Test_Approved_PLC_Functional_Test_16 := #_w1 AND #Visual_Test_Approved;
   #Reset_Functional_Test := #_w1 AND #In_Test_Parameters.Reset_PLC_Functional_Test_16;
   IF #_w1 THEN
       #Out_Functional_Test.Electrical_Current_Read_PLC_Functional_Test_16 := #Electrical_Current_Read;
   END_IF;
   #Out_Functional_Test.Life_Trigger_PLC_Functional_Test_18 := #_w1 AND #In_Functional_Test.Life_Trigger_PLC_Functional_Test_18;
   #Out_Functional_Test.Star_Test_PLC_Functional_Test_18 := #_w1 AND #In_Functional_Test.Star_Test_PLC_Functional_Test_18;
   #Out_Functional_Test.Button_PLC_Functional_Test_18 := #_w1 AND #In_Functional_Test.Button_PLC_Functional_Test_18;
   #Out_Functional_Test.Electrical_Current_Test_Approved_PLC_Functional_Test_18 := #_w1 AND #In_Functional_Test.Electrical_Current_Test_Approved_PLC_Functional_Test_18;
   #Out_Functional_Test.Visual_Test_Approved_PLC_Functional_Test_18 := #_w1 AND #In_Functional_Test.Visual_Test_Approved_PLC_Functional_Test_18;
   IF #_w1 THEN
       #Out_Functional_Test.Electrical_Current_Read_PLC_Functional_Test_18 := #In_Functional_Test.Electrical_Current_Read_PLC_Functional_Test_18;
   END_IF;
   #Out_Functional_Test.Life_Trigger_PLC_Functional_Test_20 := #_w1 AND #In_Functional_Test.Life_Trigger_PLC_Functional_Test_20;
   #Out_Functional_Test.Star_Test_PLC_Functional_Test_20 := #_w1 AND #In_Functional_Test.Star_Test_PLC_Functional_Test_20;
   #Out_Functional_Test.Button_PLC_Functional_Test_20 := #_w1 AND #In_Functional_Test.Button_PLC_Functional_Test_20;
   #Out_Functional_Test.Electrical_Current_Test_Approved_PLC_Functional_Test_20 := #_w1 AND #In_Functional_Test.Electrical_Current_Test_Approved_PLC_Functional_Test_20;
   #Out_Functional_Test.Visual_Test_Approved_PLC_Functional_Test_20 := #_w1 AND #In_Functional_Test.Visual_Test_Approved_PLC_Functional_Test_20;
   IF #_w1 THEN
       #Out_Functional_Test.Electrical_Current_Read_PLC_Functional_Test_20 := #In_Functional_Test.Electrical_Current_Read_PLC_Functional_Test_20;
   END_IF;
   #Out_Functional_Test.Life_Trigger_PLC_Functional_Test_22 := #_w1 AND #In_Functional_Test.Life_Trigger_PLC_Functional_Test_22;
   #Out_Functional_Test.Star_Test_PLC_Functional_Test_22 := #_w1 AND #In_Functional_Test.Star_Test_PLC_Functional_Test_22;
   #Out_Functional_Test.Button_PLC_Functional_Test_22 := #_w1 AND #In_Functional_Test.Button_PLC_Functional_Test_22;
   #Out_Functional_Test.Electrical_Current_Test_Approved_PLC_Functional_Test_22 := #_w1 AND #In_Functional_Test.Electrical_Current_Test_Approved_PLC_Functional_Test_22;
   #Out_Functional_Test.Visual_Test_Approved_PLC_Functional_Test_22 := #_w1 AND #In_Functional_Test.Visual_Test_Approved_PLC_Functional_Test_22;
   IF #_w1 THEN
       #Out_Functional_Test.Electrical_Current_Read_PLC_Functional_Test_22 := #In_Functional_Test.Electrical_Current_Read_PLC_Functional_Test_22;
   END_IF;
   #Out_Functional_Test.Life_Trigger_PLC_Functional_Test_24 := #_w1 AND #In_Functional_Test.Life_Trigger_PLC_Functional_Test_24;
   #Out_Functional_Test.Star_Test_PLC_Functional_Test_24 := #_w1 AND #In_Functional_Test.Star_Test_PLC_Functional_Test_24;
   #Out_Functional_Test.Button_PLC_Functional_Test_24 := #_w1 AND #In_Functional_Test.Button_PLC_Functional_Test_24;
   #Out_Functional_Test.Electrical_Current_Test_Approved_PLC_Functional_Test_24 := #_w1 AND #In_Functional_Test.Electrical_Current_Test_Approved_PLC_Functional_Test_24;
   #Out_Functional_Test.Visual_Test_Approved_PLC_Functional_Test_24 := #_w1 AND #In_Functional_Test.Visual_Test_Approved_PLC_Functional_Test_24;
   IF #_w1 THEN
       #Out_Functional_Test.Electrical_Current_Read_PLC_Functional_Test_24 := #In_Functional_Test.Electrical_Current_Read_PLC_Functional_Test_24;
   END_IF;
   #Out_Functional_Test.Life_Trigger_PLC_Functional_Test_26 := #_w1 AND #In_Functional_Test.Life_Trigger_PLC_Functional_Test_26;
   #Out_Functional_Test.Star_Test_PLC_Functional_Test_26 := #_w1 AND #In_Functional_Test.Star_Test_PLC_Functional_Test_26;
   #Out_Functional_Test.Button_PLC_Functional_Test_26 := #_w1 AND #In_Functional_Test.Button_PLC_Functional_Test_26;
   #Out_Functional_Test.Electrical_Current_Test_Approved_PLC_Functional_Test_26 := #_w1 AND #In_Functional_Test.Electrical_Current_Test_Approved_PLC_Functional_Test_26;
   #Out_Functional_Test.Visual_Test_Approved_PLC_Functional_Test_26 := #_w1 AND #In_Functional_Test.Visual_Test_Approved_PLC_Functional_Test_26;
   IF #_w1 THEN
       #Out_Functional_Test.Electrical_Current_Read_PLC_Functional_Test_26 := #In_Functional_Test.Electrical_Current_Read_PLC_Functional_Test_26;
   END_IF;
   #Out_Functional_Test.Life_Trigger_PLC_Functional_Test_28 := #_w1 AND #In_Functional_Test.Life_Trigger_PLC_Functional_Test_28;
   #Out_Functional_Test.Star_Test_PLC_Functional_Test_28 := #_w1 AND #In_Functional_Test.Star_Test_PLC_Functional_Test_28;
   #Out_Functional_Test.Button_PLC_Functional_Test_28 := #_w1 AND #In_Functional_Test.Button_PLC_Functional_Test_28;
   #Out_Functional_Test.Electrical_Current_Test_Approved_PLC_Functional_Test_28 := #_w1 AND #In_Functional_Test.Electrical_Current_Test_Approved_PLC_Functional_Test_28;
   #Out_Functional_Test.Visual_Test_Approved_PLC_Functional_Test_28 := #_w1 AND #In_Functional_Test.Visual_Test_Approved_PLC_Functional_Test_28;
   IF #_w1 THEN
       #Out_Functional_Test.Electrical_Current_Read_PLC_Functional_Test_28 := #In_Functional_Test.Electrical_Current_Read_PLC_Functional_Test_28;
   END_IF;
   #Out_Functional_Test.Life_Trigger_PLC_Functional_Test_30 := #_w1 AND #In_Functional_Test.Life_Trigger_PLC_Functional_Test_30;
   #Out_Functional_Test.Star_Test_PLC_Functional_Test_30 := #_w1 AND #In_Functional_Test.Star_Test_PLC_Functional_Test_30;
   #Out_Functional_Test.Button_PLC_Functional_Test_30 := #_w1 AND #In_Functional_Test.Button_PLC_Functional_Test_30;
   #Out_Functional_Test.Electrical_Current_Test_Approved_PLC_Functional_Test_30 := #_w1 AND #In_Functional_Test.Electrical_Current_Test_Approved_PLC_Functional_Test_30;
   #Out_Functional_Test.Visual_Test_Approved_PLC_Functional_Test_30 := #_w1 AND #In_Functional_Test.Visual_Test_Approved_PLC_Functional_Test_30;
   IF #_w1 THEN
       #Out_Functional_Test.Electrical_Current_Read_PLC_Functional_Test_30 := #In_Functional_Test.Electrical_Current_Read_PLC_Functional_Test_30;
   END_IF;
END_REGION

REGION Network 10: Functional Test Station 18
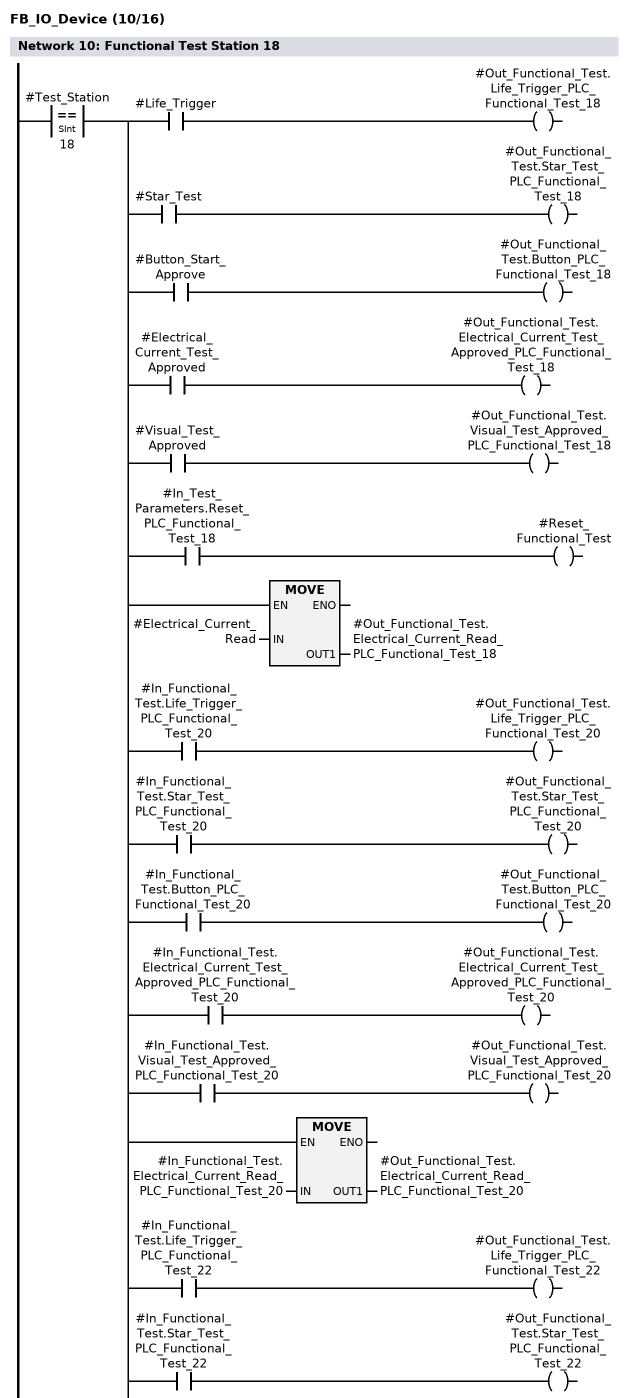
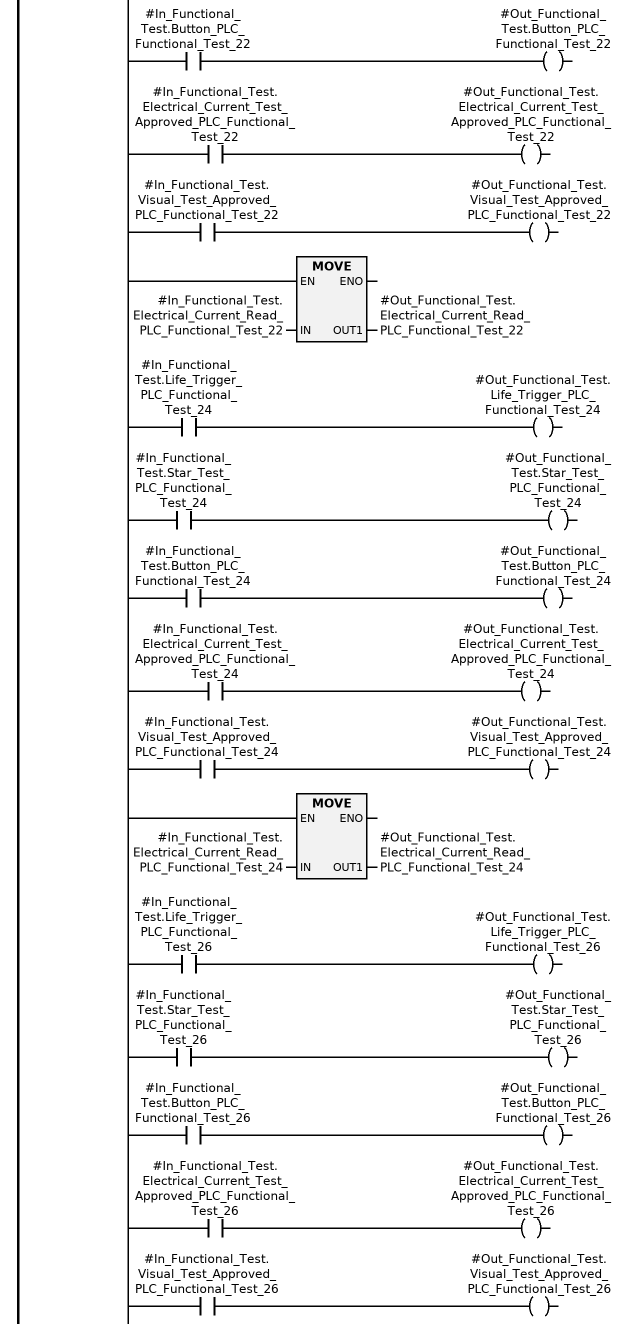
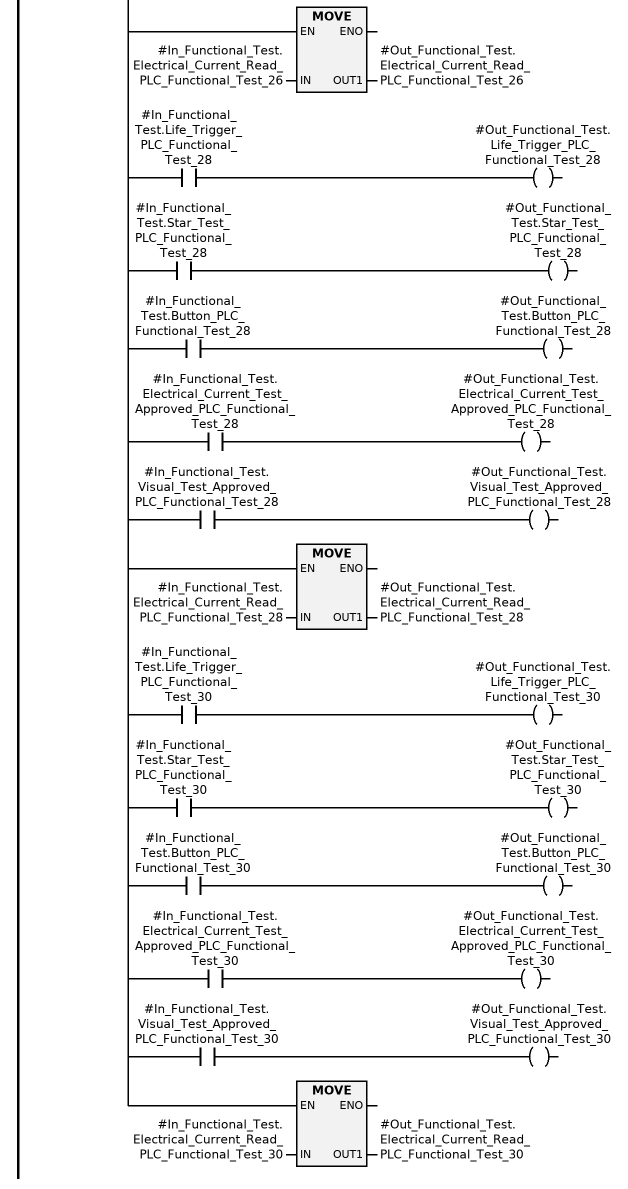
   RUNG wire#powerrail
      { S7_Templates := "SrcType := SInt" } EQ_Contact(in1 := #Test_Station, in2 := 18)
      wire#w1
      Contact( #Life_Trigger )
      Coil( #Out_Functional_Test.Life_Trigger_PLC_Functional_Test_18 )
   END_RUNG
   RUNG wire#w1
      Contact( #Star_Test )
      Coil( #Out_Functional_Test.Star_Test_PLC_Functional_Test_18 )
   END_RUNG
   RUNG wire#w1
      Contact( #Button_Start_Approve )
      Coil( #Out_Functional_Test.Button_PLC_Functional_Test_18 )
   END_RUNG
   RUNG wire#w1
      Contact( #Electrical_Current_Test_Approved )
      Coil( #Out_Functional_Test.Electrical_Current_Test_Approved_PLC_Functional_Test_18 )
   END_RUNG
   RUNG wire#w1
      Contact( #Visual_Test_Approved )
      Coil( #Out_Functional_Test.Visual_Test_Approved_PLC_Functional_Test_18 )
   END_RUNG
   RUNG wire#w1
      Contact( #In_Test_Parameters.Reset_PLC_Functional_Test_18 )
      Coil( #Reset_Functional_Test )
   END_RUNG
   RUNG wire#w1
      Move(in := #Electrical_Current_Read, out1 => #Out_Functional_Test.Electrical_Current_Read_PLC_Functional_Test_18)
   END_RUNG
   RUNG wire#w1
      Contact( #In_Functional_Test.Life_Trigger_PLC_Functional_Test_20 )
      Coil( #Out_Functional_Test.Life_Trigger_PLC_Functional_Test_20 )
   END_RUNG
   RUNG wire#w1
      Contact( #In_Functional_Test.Star_Test_PLC_Functional_Test_20 )
      Coil( #Out_Functional_Test.Star_Test_PLC_Functional_Test_20 )
   END_RUNG
   RUNG wire#w1
      Contact( #In_Functional_Test.Button_PLC_Functional_Test_20 )
      Coil( #Out_Functional_Test.Button_PLC_Functional_Test_20 )
   END_RUNG
   RUNG wire#w1
      Contact( #In_Functional_Test.Electrical_Current_Test_Approved_PLC_Functional_Test_20 )
      Coil( #Out_Functional_Test.Electrical_Current_Test_Approved_PLC_Functional_Test_20 )
   END_RUNG
   RUNG wire#w1
      Contact( #In_Functional_Test.Visual_Test_Approved_PLC_Functional_Test_20 )
      Coil( #Out_Functional_Test.Visual_Test_Approved_PLC_Functional_Test_20 )
   END_RUNG
   RUNG wire#w1
      Move(in := #In_Functional_Test.Electrical_Current_Read_PLC_Functional_Test_20, out1 => #Out_Functional_Test.Electrical_Current_Read_PLC_Functional_Test_20)
   END_RUNG
   RUNG wire#w1
      Contact( #In_Functional_Test.Life_Trigger_PLC_Functional_Test_22 )
      Coil( #Out_Functional_Test.Life_Trigger_PLC_Functional_Test_22 )
   END_RUNG
   RUNG wire#w1
      Contact( #In_Functional_Test.Star_Test_PLC_Functional_Test_22 )
      Coil( #Out_Functional_Test.Star_Test_PLC_Functional_Test_22 )
   END_RUNG
   RUNG wire#w1
      Contact( #In_Functional_Test.Button_PLC_Functional_Test_22 )
      Coil( #Out_Functional_Test.Button_PLC_Functional_Test_22 )
   END_RUNG
   RUNG wire#w1
      Contact( #In_Functional_Test.Electrical_Current_Test_Approved_PLC_Functional_Test_22 )
      Coil( #Out_Functional_Test.Electrical_Current_Test_Approved_PLC_Functional_Test_22 )
   END_RUNG
   RUNG wire#w1
      Contact( #In_Functional_Test.Visual_Test_Approved_PLC_Functional_Test_22 )
      Coil( #Out_Functional_Test.Visual_Test_Approved_PLC_Functional_Test_22 )
   END_RUNG
   RUNG wire#w1
      Move(in := #In_Functional_Test.Electrical_Current_Read_PLC_Functional_Test_22, out1 => #Out_Functional_Test.Electrical_Current_Read_PLC_Functional_Test_22)
   END_RUNG
   RUNG wire#w1
      Contact( #In_Functional_Test.Life_Trigger_PLC_Functional_Test_24 )
      Coil( #Out_Functional_Test.Life_Trigger_PLC_Functional_Test_24 )
   END_RUNG
   RUNG wire#w1
      Contact( #In_Functional_Test.Star_Test_PLC_Functional_Test_24 )
      Coil( #Out_Functional_Test.Star_Test_PLC_Functional_Test_24 )
   END_RUNG
   RUNG wire#w1
      Contact( #In_Functional_Test.Button_PLC_Functional_Test_24 )
      Coil( #Out_Functional_Test.Button_PLC_Functional_Test_24 )
   END_RUNG
   RUNG wire#w1
      Contact( #In_Functional_Test.Electrical_Current_Test_Approved_PLC_Functional_Test_24 )
      Coil( #Out_Functional_Test.Electrical_Current_Test_Approved_PLC_Functional_Test_24 )
   END_RUNG
   RUNG wire#w1
      Contact( #In_Functional_Test.Visual_Test_Approved_PLC_Functional_Test_24 )
      Coil( #Out_Functional_Test.Visual_Test_Approved_PLC_Functional_Test_24 )
   END_RUNG
   RUNG wire#w1
      Move(in := #In_Functional_Test.Electrical_Current_Read_PLC_Functional_Test_24, out1 => #Out_Functional_Test.Electrical_Current_Read_PLC_Functional_Test_24)
   END_RUNG
   RUNG wire#w1
      Contact( #In_Functional_Test.Life_Trigger_PLC_Functional_Test_26 )
      Coil( #Out_Functional_Test.Life_Trigger_PLC_Functional_Test_26 )
   END_RUNG
   RUNG wire#w1
      Contact( #In_Functional_Test.Star_Test_PLC_Functional_Test_26 )
      Coil( #Out_Functional_Test.Star_Test_PLC_Functional_Test_26 )
   END_RUNG
   RUNG wire#w1
      Contact( #In_Functional_Test.Button_PLC_Functional_Test_26 )
      Coil( #Out_Functional_Test.Button_PLC_Functional_Test_26 )
   END_RUNG
   RUNG wire#w1
      Contact( #In_Functional_Test.Electrical_Current_Test_Approved_PLC_Functional_Test_26 )
      Coil( #Out_Functional_Test.Electrical_Current_Test_Approved_PLC_Functional_Test_26 )
   END_RUNG
   RUNG wire#w1
      Contact( #In_Functional_Test.Visual_Test_Approved_PLC_Functional_Test_26 )
      Coil( #Out_Functional_Test.Visual_Test_Approved_PLC_Functional_Test_26 )
   END_RUNG
   RUNG wire#w1
      Move(in := #In_Functional_Test.Electrical_Current_Read_PLC_Functional_Test_26, out1 => #Out_Functional_Test.Electrical_Current_Read_PLC_Functional_Test_26)
   END_RUNG
   RUNG wire#w1
      Contact( #In_Functional_Test.Life_Trigger_PLC_Functional_Test_28 )
      Coil( #Out_Functional_Test.Life_Trigger_PLC_Functional_Test_28 )
   END_RUNG
   RUNG wire#w1
      Contact( #In_Functional_Test.Star_Test_PLC_Functional_Test_28 )
      Coil( #Out_Functional_Test.Star_Test_PLC_Functional_Test_28 )
   END_RUNG
   RUNG wire#w1
      Contact( #In_Functional_Test.Button_PLC_Functional_Test_28 )
      Coil( #Out_Functional_Test.Button_PLC_Functional_Test_28 )
   END_RUNG
   RUNG wire#w1
      Contact( #In_Functional_Test.Electrical_Current_Test_Approved_PLC_Functional_Test_28 )
      Coil( #Out_Functional_Test.Electrical_Current_Test_Approved_PLC_Functional_Test_28 )
   END_RUNG
   RUNG wire#w1
      Contact( #In_Functional_Test.Visual_Test_Approved_PLC_Functional_Test_28 )
      Coil( #Out_Functional_Test.Visual_Test_Approved_PLC_Functional_Test_28 )
   END_RUNG
   RUNG wire#w1
      Move(in := #In_Functional_Test.Electrical_Current_Read_PLC_Functional_Test_28, out1 => #Out_Functional_Test.Electrical_Current_Read_PLC_Functional_Test_28)
   END_RUNG
   RUNG wire#w1
      Contact( #In_Functional_Test.Life_Trigger_PLC_Functional_Test_30 )
      Coil( #Out_Functional_Test.Life_Trigger_PLC_Functional_Test_30 )
   END_RUNG
   RUNG wire#w1
      Contact( #In_Functional_Test.Star_Test_PLC_Functional_Test_30 )
      Coil( #Out_Functional_Test.Star_Test_PLC_Functional_Test_30 )
   END_RUNG
   RUNG wire#w1
      Contact( #In_Functional_Test.Button_PLC_Functional_Test_30 )
      Coil( #Out_Functional_Test.Button_PLC_Functional_Test_30 )
   END_RUNG
   RUNG wire#w1
      Contact( #In_Functional_Test.Electrical_Current_Test_Approved_PLC_Functional_Test_30 )
      Coil( #Out_Functional_Test.Electrical_Current_Test_Approved_PLC_Functional_Test_30 )
   END_RUNG
   RUNG wire#w1
      Contact( #In_Functional_Test.Visual_Test_Approved_PLC_Functional_Test_30 )
      Coil( #Out_Functional_Test.Visual_Test_Approved_PLC_Functional_Test_30 )
   END_RUNG
   RUNG wire#w1
      Move(in := #In_Functional_Test.Electrical_Current_Read_PLC_Functional_Test_30, out1 => #Out_Functional_Test.Electrical_Current_Read_PLC_Functional_Test_30)
   END_RUNG
   // the same network as SCL:
   #_w1 := #Test_Station = 18;
   #Out_Functional_Test.Life_Trigger_PLC_Functional_Test_18 := #_w1 AND #Life_Trigger;
   #Out_Functional_Test.Star_Test_PLC_Functional_Test_18 := #_w1 AND #Star_Test;
   #Out_Functional_Test.Button_PLC_Functional_Test_18 := #_w1 AND #Button_Start_Approve;
   #Out_Functional_Test.Electrical_Current_Test_Approved_PLC_Functional_Test_18 := #_w1 AND #Electrical_Current_Test_Approved;
   #Out_Functional_Test.Visual_Test_Approved_PLC_Functional_Test_18 := #_w1 AND #Visual_Test_Approved;
   #Reset_Functional_Test := #_w1 AND #In_Test_Parameters.Reset_PLC_Functional_Test_18;
   IF #_w1 THEN
       #Out_Functional_Test.Electrical_Current_Read_PLC_Functional_Test_18 := #Electrical_Current_Read;
   END_IF;
   #Out_Functional_Test.Life_Trigger_PLC_Functional_Test_20 := #_w1 AND #In_Functional_Test.Life_Trigger_PLC_Functional_Test_20;
   #Out_Functional_Test.Star_Test_PLC_Functional_Test_20 := #_w1 AND #In_Functional_Test.Star_Test_PLC_Functional_Test_20;
   #Out_Functional_Test.Button_PLC_Functional_Test_20 := #_w1 AND #In_Functional_Test.Button_PLC_Functional_Test_20;
   #Out_Functional_Test.Electrical_Current_Test_Approved_PLC_Functional_Test_20 := #_w1 AND #In_Functional_Test.Electrical_Current_Test_Approved_PLC_Functional_Test_20;
   #Out_Functional_Test.Visual_Test_Approved_PLC_Functional_Test_20 := #_w1 AND #In_Functional_Test.Visual_Test_Approved_PLC_Functional_Test_20;
   IF #_w1 THEN
       #Out_Functional_Test.Electrical_Current_Read_PLC_Functional_Test_20 := #In_Functional_Test.Electrical_Current_Read_PLC_Functional_Test_20;
   END_IF;
   #Out_Functional_Test.Life_Trigger_PLC_Functional_Test_22 := #_w1 AND #In_Functional_Test.Life_Trigger_PLC_Functional_Test_22;
   #Out_Functional_Test.Star_Test_PLC_Functional_Test_22 := #_w1 AND #In_Functional_Test.Star_Test_PLC_Functional_Test_22;
   #Out_Functional_Test.Button_PLC_Functional_Test_22 := #_w1 AND #In_Functional_Test.Button_PLC_Functional_Test_22;
   #Out_Functional_Test.Electrical_Current_Test_Approved_PLC_Functional_Test_22 := #_w1 AND #In_Functional_Test.Electrical_Current_Test_Approved_PLC_Functional_Test_22;
   #Out_Functional_Test.Visual_Test_Approved_PLC_Functional_Test_22 := #_w1 AND #In_Functional_Test.Visual_Test_Approved_PLC_Functional_Test_22;
   IF #_w1 THEN
       #Out_Functional_Test.Electrical_Current_Read_PLC_Functional_Test_22 := #In_Functional_Test.Electrical_Current_Read_PLC_Functional_Test_22;
   END_IF;
   #Out_Functional_Test.Life_Trigger_PLC_Functional_Test_24 := #_w1 AND #In_Functional_Test.Life_Trigger_PLC_Functional_Test_24;
   #Out_Functional_Test.Star_Test_PLC_Functional_Test_24 := #_w1 AND #In_Functional_Test.Star_Test_PLC_Functional_Test_24;
   #Out_Functional_Test.Button_PLC_Functional_Test_24 := #_w1 AND #In_Functional_Test.Button_PLC_Functional_Test_24;
   #Out_Functional_Test.Electrical_Current_Test_Approved_PLC_Functional_Test_24 := #_w1 AND #In_Functional_Test.Electrical_Current_Test_Approved_PLC_Functional_Test_24;
   #Out_Functional_Test.Visual_Test_Approved_PLC_Functional_Test_24 := #_w1 AND #In_Functional_Test.Visual_Test_Approved_PLC_Functional_Test_24;
   IF #_w1 THEN
       #Out_Functional_Test.Electrical_Current_Read_PLC_Functional_Test_24 := #In_Functional_Test.Electrical_Current_Read_PLC_Functional_Test_24;
   END_IF;
   #Out_Functional_Test.Life_Trigger_PLC_Functional_Test_26 := #_w1 AND #In_Functional_Test.Life_Trigger_PLC_Functional_Test_26;
   #Out_Functional_Test.Star_Test_PLC_Functional_Test_26 := #_w1 AND #In_Functional_Test.Star_Test_PLC_Functional_Test_26;
   #Out_Functional_Test.Button_PLC_Functional_Test_26 := #_w1 AND #In_Functional_Test.Button_PLC_Functional_Test_26;
   #Out_Functional_Test.Electrical_Current_Test_Approved_PLC_Functional_Test_26 := #_w1 AND #In_Functional_Test.Electrical_Current_Test_Approved_PLC_Functional_Test_26;
   #Out_Functional_Test.Visual_Test_Approved_PLC_Functional_Test_26 := #_w1 AND #In_Functional_Test.Visual_Test_Approved_PLC_Functional_Test_26;
   IF #_w1 THEN
       #Out_Functional_Test.Electrical_Current_Read_PLC_Functional_Test_26 := #In_Functional_Test.Electrical_Current_Read_PLC_Functional_Test_26;
   END_IF;
   #Out_Functional_Test.Life_Trigger_PLC_Functional_Test_28 := #_w1 AND #In_Functional_Test.Life_Trigger_PLC_Functional_Test_28;
   #Out_Functional_Test.Star_Test_PLC_Functional_Test_28 := #_w1 AND #In_Functional_Test.Star_Test_PLC_Functional_Test_28;
   #Out_Functional_Test.Button_PLC_Functional_Test_28 := #_w1 AND #In_Functional_Test.Button_PLC_Functional_Test_28;
   #Out_Functional_Test.Electrical_Current_Test_Approved_PLC_Functional_Test_28 := #_w1 AND #In_Functional_Test.Electrical_Current_Test_Approved_PLC_Functional_Test_28;
   #Out_Functional_Test.Visual_Test_Approved_PLC_Functional_Test_28 := #_w1 AND #In_Functional_Test.Visual_Test_Approved_PLC_Functional_Test_28;
   IF #_w1 THEN
       #Out_Functional_Test.Electrical_Current_Read_PLC_Functional_Test_28 := #In_Functional_Test.Electrical_Current_Read_PLC_Functional_Test_28;
   END_IF;
   #Out_Functional_Test.Life_Trigger_PLC_Functional_Test_30 := #_w1 AND #In_Functional_Test.Life_Trigger_PLC_Functional_Test_30;
   #Out_Functional_Test.Star_Test_PLC_Functional_Test_30 := #_w1 AND #In_Functional_Test.Star_Test_PLC_Functional_Test_30;
   #Out_Functional_Test.Button_PLC_Functional_Test_30 := #_w1 AND #In_Functional_Test.Button_PLC_Functional_Test_30;
   #Out_Functional_Test.Electrical_Current_Test_Approved_PLC_Functional_Test_30 := #_w1 AND #In_Functional_Test.Electrical_Current_Test_Approved_PLC_Functional_Test_30;
   #Out_Functional_Test.Visual_Test_Approved_PLC_Functional_Test_30 := #_w1 AND #In_Functional_Test.Visual_Test_Approved_PLC_Functional_Test_30;
   IF #_w1 THEN
       #Out_Functional_Test.Electrical_Current_Read_PLC_Functional_Test_30 := #In_Functional_Test.Electrical_Current_Read_PLC_Functional_Test_30;
   END_IF;
END_REGION

REGION Network 11: Functional Test Station 20
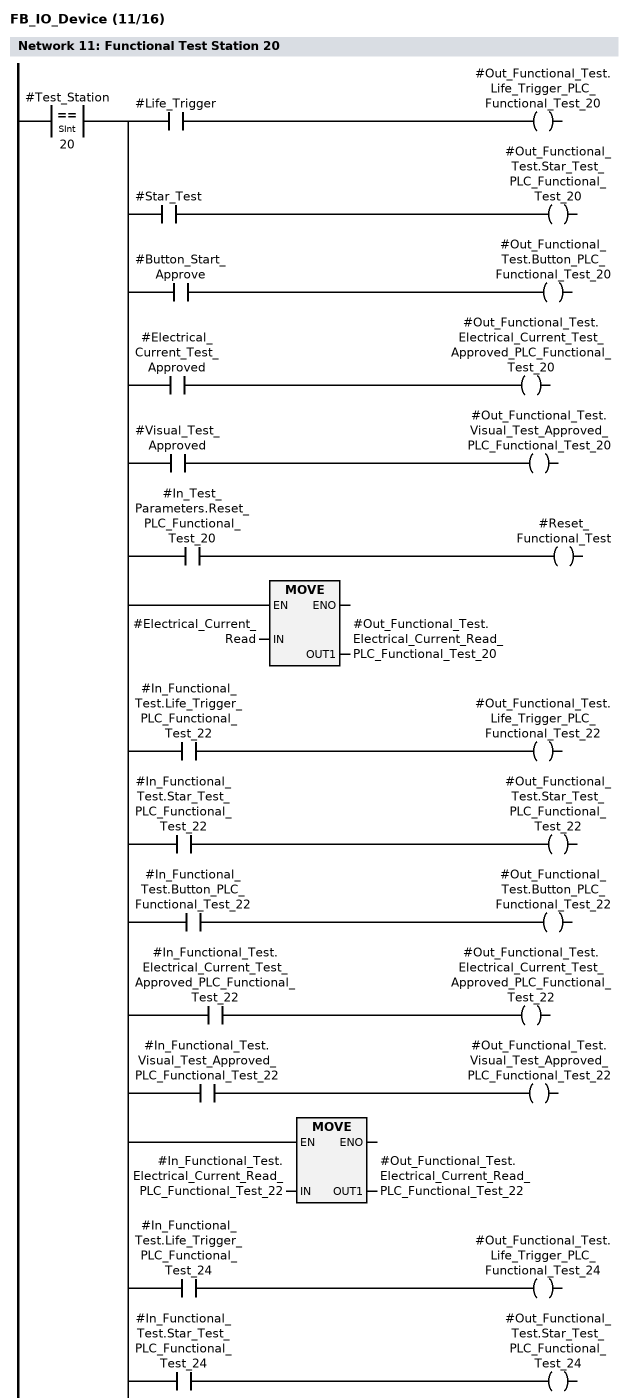
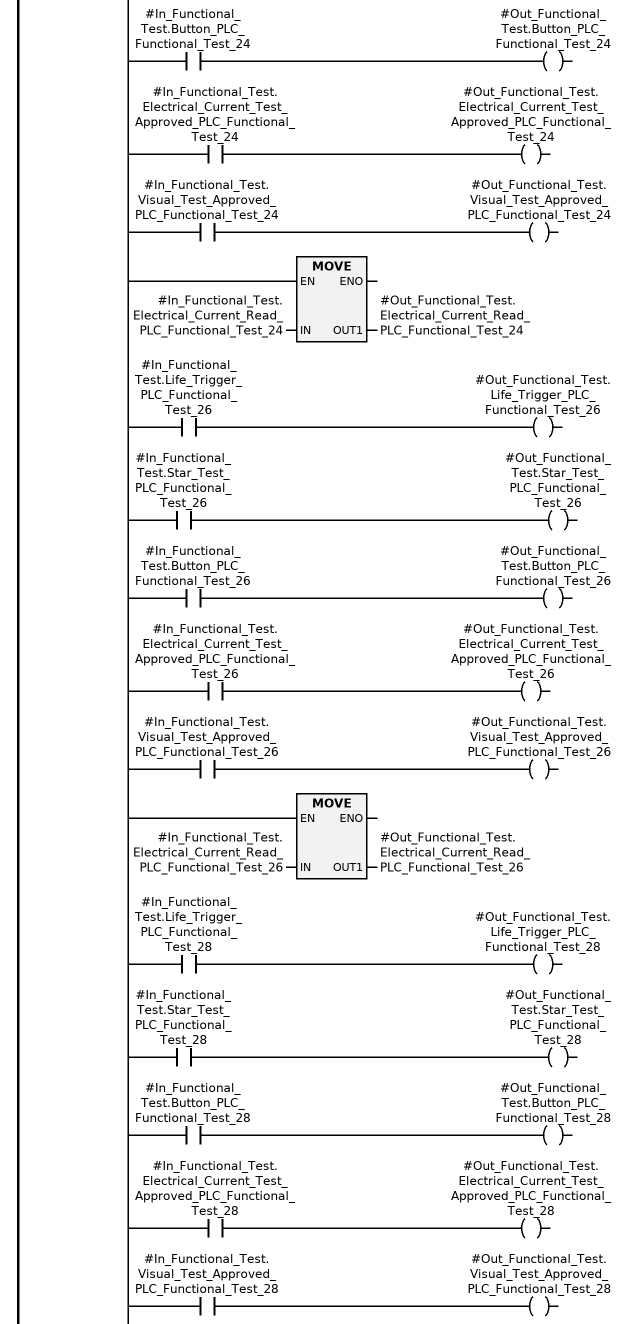
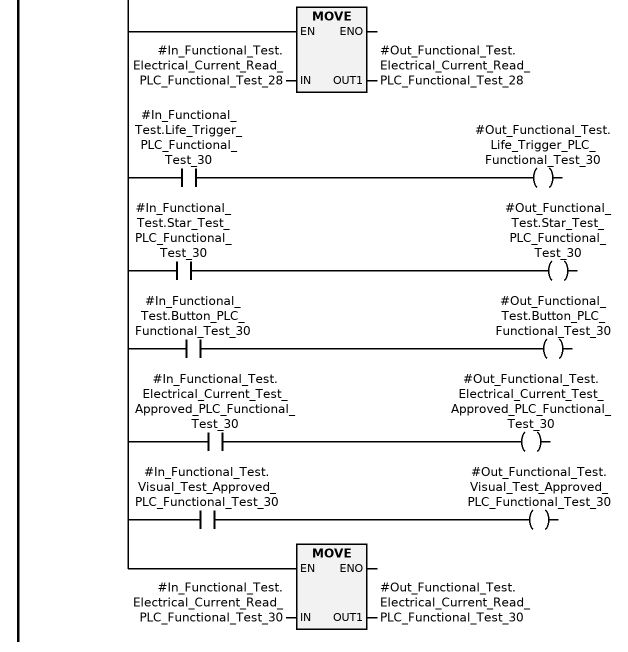
   RUNG wire#powerrail
      { S7_Templates := "SrcType := SInt" } EQ_Contact(in1 := #Test_Station, in2 := 20)
      wire#w1
      Contact( #Life_Trigger )
      Coil( #Out_Functional_Test.Life_Trigger_PLC_Functional_Test_20 )
   END_RUNG
   RUNG wire#w1
      Contact( #Star_Test )
      Coil( #Out_Functional_Test.Star_Test_PLC_Functional_Test_20 )
   END_RUNG
   RUNG wire#w1
      Contact( #Button_Start_Approve )
      Coil( #Out_Functional_Test.Button_PLC_Functional_Test_20 )
   END_RUNG
   RUNG wire#w1
      Contact( #Electrical_Current_Test_Approved )
      Coil( #Out_Functional_Test.Electrical_Current_Test_Approved_PLC_Functional_Test_20 )
   END_RUNG
   RUNG wire#w1
      Contact( #Visual_Test_Approved )
      Coil( #Out_Functional_Test.Visual_Test_Approved_PLC_Functional_Test_20 )
   END_RUNG
   RUNG wire#w1
      Contact( #In_Test_Parameters.Reset_PLC_Functional_Test_20 )
      Coil( #Reset_Functional_Test )
   END_RUNG
   RUNG wire#w1
      Move(in := #Electrical_Current_Read, out1 => #Out_Functional_Test.Electrical_Current_Read_PLC_Functional_Test_20)
   END_RUNG
   RUNG wire#w1
      Contact( #In_Functional_Test.Life_Trigger_PLC_Functional_Test_22 )
      Coil( #Out_Functional_Test.Life_Trigger_PLC_Functional_Test_22 )
   END_RUNG
   RUNG wire#w1
      Contact( #In_Functional_Test.Star_Test_PLC_Functional_Test_22 )
      Coil( #Out_Functional_Test.Star_Test_PLC_Functional_Test_22 )
   END_RUNG
   RUNG wire#w1
      Contact( #In_Functional_Test.Button_PLC_Functional_Test_22 )
      Coil( #Out_Functional_Test.Button_PLC_Functional_Test_22 )
   END_RUNG
   RUNG wire#w1
      Contact( #In_Functional_Test.Electrical_Current_Test_Approved_PLC_Functional_Test_22 )
      Coil( #Out_Functional_Test.Electrical_Current_Test_Approved_PLC_Functional_Test_22 )
   END_RUNG
   RUNG wire#w1
      Contact( #In_Functional_Test.Visual_Test_Approved_PLC_Functional_Test_22 )
      Coil( #Out_Functional_Test.Visual_Test_Approved_PLC_Functional_Test_22 )
   END_RUNG
   RUNG wire#w1
      Move(in := #In_Functional_Test.Electrical_Current_Read_PLC_Functional_Test_22, out1 => #Out_Functional_Test.Electrical_Current_Read_PLC_Functional_Test_22)
   END_RUNG
   RUNG wire#w1
      Contact( #In_Functional_Test.Life_Trigger_PLC_Functional_Test_24 )
      Coil( #Out_Functional_Test.Life_Trigger_PLC_Functional_Test_24 )
   END_RUNG
   RUNG wire#w1
      Contact( #In_Functional_Test.Star_Test_PLC_Functional_Test_24 )
      Coil( #Out_Functional_Test.Star_Test_PLC_Functional_Test_24 )
   END_RUNG
   RUNG wire#w1
      Contact( #In_Functional_Test.Button_PLC_Functional_Test_24 )
      Coil( #Out_Functional_Test.Button_PLC_Functional_Test_24 )
   END_RUNG
   RUNG wire#w1
      Contact( #In_Functional_Test.Electrical_Current_Test_Approved_PLC_Functional_Test_24 )
      Coil( #Out_Functional_Test.Electrical_Current_Test_Approved_PLC_Functional_Test_24 )
   END_RUNG
   RUNG wire#w1
      Contact( #In_Functional_Test.Visual_Test_Approved_PLC_Functional_Test_24 )
      Coil( #Out_Functional_Test.Visual_Test_Approved_PLC_Functional_Test_24 )
   END_RUNG
   RUNG wire#w1
      Move(in := #In_Functional_Test.Electrical_Current_Read_PLC_Functional_Test_24, out1 => #Out_Functional_Test.Electrical_Current_Read_PLC_Functional_Test_24)
   END_RUNG
   RUNG wire#w1
      Contact( #In_Functional_Test.Life_Trigger_PLC_Functional_Test_26 )
      Coil( #Out_Functional_Test.Life_Trigger_PLC_Functional_Test_26 )
   END_RUNG
   RUNG wire#w1
      Contact( #In_Functional_Test.Star_Test_PLC_Functional_Test_26 )
      Coil( #Out_Functional_Test.Star_Test_PLC_Functional_Test_26 )
   END_RUNG
   RUNG wire#w1
      Contact( #In_Functional_Test.Button_PLC_Functional_Test_26 )
      Coil( #Out_Functional_Test.Button_PLC_Functional_Test_26 )
   END_RUNG
   RUNG wire#w1
      Contact( #In_Functional_Test.Electrical_Current_Test_Approved_PLC_Functional_Test_26 )
      Coil( #Out_Functional_Test.Electrical_Current_Test_Approved_PLC_Functional_Test_26 )
   END_RUNG
   RUNG wire#w1
      Contact( #In_Functional_Test.Visual_Test_Approved_PLC_Functional_Test_26 )
      Coil( #Out_Functional_Test.Visual_Test_Approved_PLC_Functional_Test_26 )
   END_RUNG
   RUNG wire#w1
      Move(in := #In_Functional_Test.Electrical_Current_Read_PLC_Functional_Test_26, out1 => #Out_Functional_Test.Electrical_Current_Read_PLC_Functional_Test_26)
   END_RUNG
   RUNG wire#w1
      Contact( #In_Functional_Test.Life_Trigger_PLC_Functional_Test_28 )
      Coil( #Out_Functional_Test.Life_Trigger_PLC_Functional_Test_28 )
   END_RUNG
   RUNG wire#w1
      Contact( #In_Functional_Test.Star_Test_PLC_Functional_Test_28 )
      Coil( #Out_Functional_Test.Star_Test_PLC_Functional_Test_28 )
   END_RUNG
   RUNG wire#w1
      Contact( #In_Functional_Test.Button_PLC_Functional_Test_28 )
      Coil( #Out_Functional_Test.Button_PLC_Functional_Test_28 )
   END_RUNG
   RUNG wire#w1
      Contact( #In_Functional_Test.Electrical_Current_Test_Approved_PLC_Functional_Test_28 )
      Coil( #Out_Functional_Test.Electrical_Current_Test_Approved_PLC_Functional_Test_28 )
   END_RUNG
   RUNG wire#w1
      Contact( #In_Functional_Test.Visual_Test_Approved_PLC_Functional_Test_28 )
      Coil( #Out_Functional_Test.Visual_Test_Approved_PLC_Functional_Test_28 )
   END_RUNG
   RUNG wire#w1
      Move(in := #In_Functional_Test.Electrical_Current_Read_PLC_Functional_Test_28, out1 => #Out_Functional_Test.Electrical_Current_Read_PLC_Functional_Test_28)
   END_RUNG
   RUNG wire#w1
      Contact( #In_Functional_Test.Life_Trigger_PLC_Functional_Test_30 )
      Coil( #Out_Functional_Test.Life_Trigger_PLC_Functional_Test_30 )
   END_RUNG
   RUNG wire#w1
      Contact( #In_Functional_Test.Star_Test_PLC_Functional_Test_30 )
      Coil( #Out_Functional_Test.Star_Test_PLC_Functional_Test_30 )
   END_RUNG
   RUNG wire#w1
      Contact( #In_Functional_Test.Button_PLC_Functional_Test_30 )
      Coil( #Out_Functional_Test.Button_PLC_Functional_Test_30 )
   END_RUNG
   RUNG wire#w1
      Contact( #In_Functional_Test.Electrical_Current_Test_Approved_PLC_Functional_Test_30 )
      Coil( #Out_Functional_Test.Electrical_Current_Test_Approved_PLC_Functional_Test_30 )
   END_RUNG
   RUNG wire#w1
      Contact( #In_Functional_Test.Visual_Test_Approved_PLC_Functional_Test_30 )
      Coil( #Out_Functional_Test.Visual_Test_Approved_PLC_Functional_Test_30 )
   END_RUNG
   RUNG wire#w1
      Move(in := #In_Functional_Test.Electrical_Current_Read_PLC_Functional_Test_30, out1 => #Out_Functional_Test.Electrical_Current_Read_PLC_Functional_Test_30)
   END_RUNG
   // the same network as SCL:
   #_w1 := #Test_Station = 20;
   #Out_Functional_Test.Life_Trigger_PLC_Functional_Test_20 := #_w1 AND #Life_Trigger;
   #Out_Functional_Test.Star_Test_PLC_Functional_Test_20 := #_w1 AND #Star_Test;
   #Out_Functional_Test.Button_PLC_Functional_Test_20 := #_w1 AND #Button_Start_Approve;
   #Out_Functional_Test.Electrical_Current_Test_Approved_PLC_Functional_Test_20 := #_w1 AND #Electrical_Current_Test_Approved;
   #Out_Functional_Test.Visual_Test_Approved_PLC_Functional_Test_20 := #_w1 AND #Visual_Test_Approved;
   #Reset_Functional_Test := #_w1 AND #In_Test_Parameters.Reset_PLC_Functional_Test_20;
   IF #_w1 THEN
       #Out_Functional_Test.Electrical_Current_Read_PLC_Functional_Test_20 := #Electrical_Current_Read;
   END_IF;
   #Out_Functional_Test.Life_Trigger_PLC_Functional_Test_22 := #_w1 AND #In_Functional_Test.Life_Trigger_PLC_Functional_Test_22;
   #Out_Functional_Test.Star_Test_PLC_Functional_Test_22 := #_w1 AND #In_Functional_Test.Star_Test_PLC_Functional_Test_22;
   #Out_Functional_Test.Button_PLC_Functional_Test_22 := #_w1 AND #In_Functional_Test.Button_PLC_Functional_Test_22;
   #Out_Functional_Test.Electrical_Current_Test_Approved_PLC_Functional_Test_22 := #_w1 AND #In_Functional_Test.Electrical_Current_Test_Approved_PLC_Functional_Test_22;
   #Out_Functional_Test.Visual_Test_Approved_PLC_Functional_Test_22 := #_w1 AND #In_Functional_Test.Visual_Test_Approved_PLC_Functional_Test_22;
   IF #_w1 THEN
       #Out_Functional_Test.Electrical_Current_Read_PLC_Functional_Test_22 := #In_Functional_Test.Electrical_Current_Read_PLC_Functional_Test_22;
   END_IF;
   #Out_Functional_Test.Life_Trigger_PLC_Functional_Test_24 := #_w1 AND #In_Functional_Test.Life_Trigger_PLC_Functional_Test_24;
   #Out_Functional_Test.Star_Test_PLC_Functional_Test_24 := #_w1 AND #In_Functional_Test.Star_Test_PLC_Functional_Test_24;
   #Out_Functional_Test.Button_PLC_Functional_Test_24 := #_w1 AND #In_Functional_Test.Button_PLC_Functional_Test_24;
   #Out_Functional_Test.Electrical_Current_Test_Approved_PLC_Functional_Test_24 := #_w1 AND #In_Functional_Test.Electrical_Current_Test_Approved_PLC_Functional_Test_24;
   #Out_Functional_Test.Visual_Test_Approved_PLC_Functional_Test_24 := #_w1 AND #In_Functional_Test.Visual_Test_Approved_PLC_Functional_Test_24;
   IF #_w1 THEN
       #Out_Functional_Test.Electrical_Current_Read_PLC_Functional_Test_24 := #In_Functional_Test.Electrical_Current_Read_PLC_Functional_Test_24;
   END_IF;
   #Out_Functional_Test.Life_Trigger_PLC_Functional_Test_26 := #_w1 AND #In_Functional_Test.Life_Trigger_PLC_Functional_Test_26;
   #Out_Functional_Test.Star_Test_PLC_Functional_Test_26 := #_w1 AND #In_Functional_Test.Star_Test_PLC_Functional_Test_26;
   #Out_Functional_Test.Button_PLC_Functional_Test_26 := #_w1 AND #In_Functional_Test.Button_PLC_Functional_Test_26;
   #Out_Functional_Test.Electrical_Current_Test_Approved_PLC_Functional_Test_26 := #_w1 AND #In_Functional_Test.Electrical_Current_Test_Approved_PLC_Functional_Test_26;
   #Out_Functional_Test.Visual_Test_Approved_PLC_Functional_Test_26 := #_w1 AND #In_Functional_Test.Visual_Test_Approved_PLC_Functional_Test_26;
   IF #_w1 THEN
       #Out_Functional_Test.Electrical_Current_Read_PLC_Functional_Test_26 := #In_Functional_Test.Electrical_Current_Read_PLC_Functional_Test_26;
   END_IF;
   #Out_Functional_Test.Life_Trigger_PLC_Functional_Test_28 := #_w1 AND #In_Functional_Test.Life_Trigger_PLC_Functional_Test_28;
   #Out_Functional_Test.Star_Test_PLC_Functional_Test_28 := #_w1 AND #In_Functional_Test.Star_Test_PLC_Functional_Test_28;
   #Out_Functional_Test.Button_PLC_Functional_Test_28 := #_w1 AND #In_Functional_Test.Button_PLC_Functional_Test_28;
   #Out_Functional_Test.Electrical_Current_Test_Approved_PLC_Functional_Test_28 := #_w1 AND #In_Functional_Test.Electrical_Current_Test_Approved_PLC_Functional_Test_28;
   #Out_Functional_Test.Visual_Test_Approved_PLC_Functional_Test_28 := #_w1 AND #In_Functional_Test.Visual_Test_Approved_PLC_Functional_Test_28;
   IF #_w1 THEN
       #Out_Functional_Test.Electrical_Current_Read_PLC_Functional_Test_28 := #In_Functional_Test.Electrical_Current_Read_PLC_Functional_Test_28;
   END_IF;
   #Out_Functional_Test.Life_Trigger_PLC_Functional_Test_30 := #_w1 AND #In_Functional_Test.Life_Trigger_PLC_Functional_Test_30;
   #Out_Functional_Test.Star_Test_PLC_Functional_Test_30 := #_w1 AND #In_Functional_Test.Star_Test_PLC_Functional_Test_30;
   #Out_Functional_Test.Button_PLC_Functional_Test_30 := #_w1 AND #In_Functional_Test.Button_PLC_Functional_Test_30;
   #Out_Functional_Test.Electrical_Current_Test_Approved_PLC_Functional_Test_30 := #_w1 AND #In_Functional_Test.Electrical_Current_Test_Approved_PLC_Functional_Test_30;
   #Out_Functional_Test.Visual_Test_Approved_PLC_Functional_Test_30 := #_w1 AND #In_Functional_Test.Visual_Test_Approved_PLC_Functional_Test_30;
   IF #_w1 THEN
       #Out_Functional_Test.Electrical_Current_Read_PLC_Functional_Test_30 := #In_Functional_Test.Electrical_Current_Read_PLC_Functional_Test_30;
   END_IF;
END_REGION

REGION Network 12: Functional Test Station 22
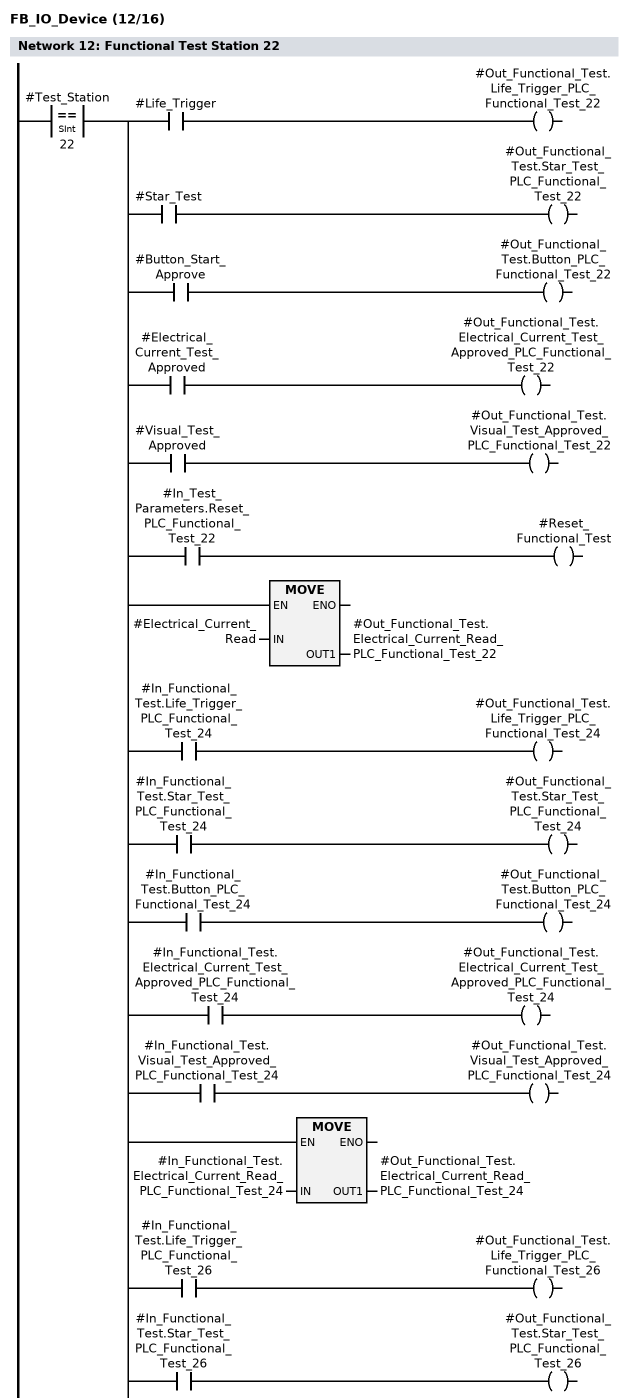
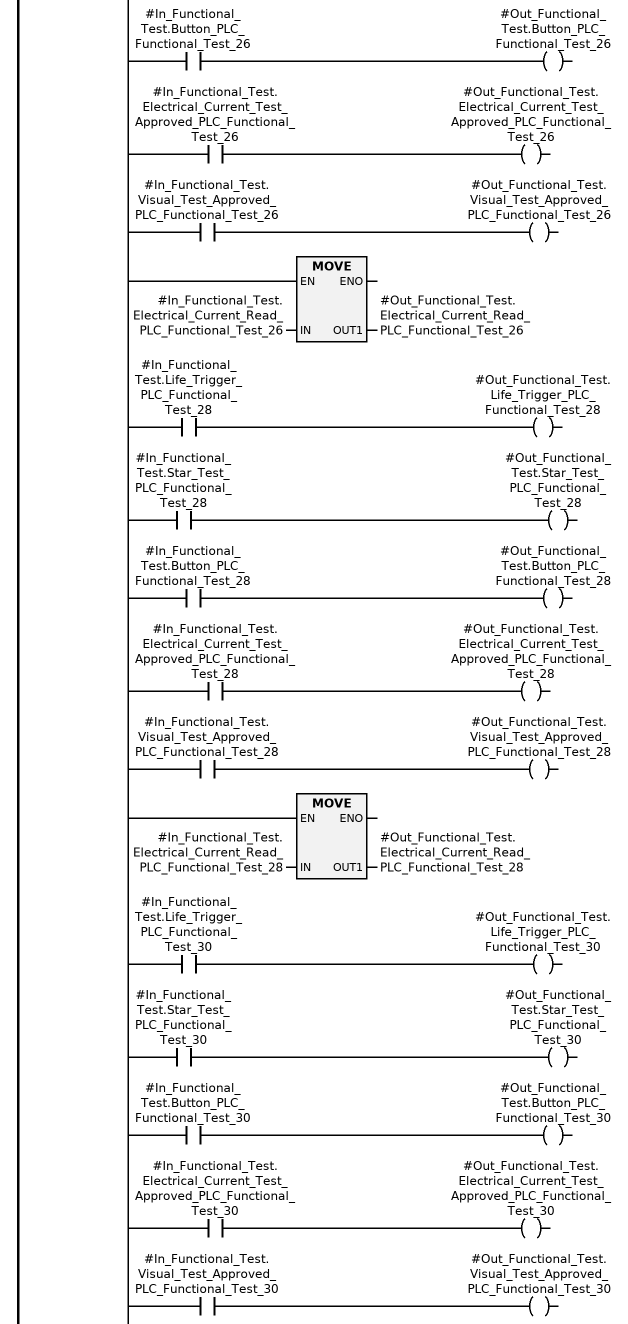
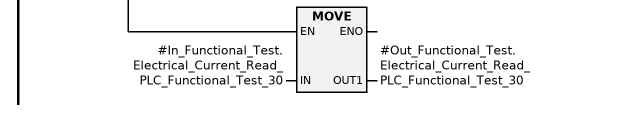
   RUNG wire#powerrail
      { S7_Templates := "SrcType := SInt" } EQ_Contact(in1 := #Test_Station, in2 := 22)
      wire#w1
      Contact( #Life_Trigger )
      Coil( #Out_Functional_Test.Life_Trigger_PLC_Functional_Test_22 )
   END_RUNG
   RUNG wire#w1
      Contact( #Star_Test )
      Coil( #Out_Functional_Test.Star_Test_PLC_Functional_Test_22 )
   END_RUNG
   RUNG wire#w1
      Contact( #Button_Start_Approve )
      Coil( #Out_Functional_Test.Button_PLC_Functional_Test_22 )
   END_RUNG
   RUNG wire#w1
      Contact( #Electrical_Current_Test_Approved )
      Coil( #Out_Functional_Test.Electrical_Current_Test_Approved_PLC_Functional_Test_22 )
   END_RUNG
   RUNG wire#w1
      Contact( #Visual_Test_Approved )
      Coil( #Out_Functional_Test.Visual_Test_Approved_PLC_Functional_Test_22 )
   END_RUNG
   RUNG wire#w1
      Contact( #In_Test_Parameters.Reset_PLC_Functional_Test_22 )
      Coil( #Reset_Functional_Test )
   END_RUNG
   RUNG wire#w1
      Move(in := #Electrical_Current_Read, out1 => #Out_Functional_Test.Electrical_Current_Read_PLC_Functional_Test_22)
   END_RUNG
   RUNG wire#w1
      Contact( #In_Functional_Test.Life_Trigger_PLC_Functional_Test_24 )
      Coil( #Out_Functional_Test.Life_Trigger_PLC_Functional_Test_24 )
   END_RUNG
   RUNG wire#w1
      Contact( #In_Functional_Test.Star_Test_PLC_Functional_Test_24 )
      Coil( #Out_Functional_Test.Star_Test_PLC_Functional_Test_24 )
   END_RUNG
   RUNG wire#w1
      Contact( #In_Functional_Test.Button_PLC_Functional_Test_24 )
      Coil( #Out_Functional_Test.Button_PLC_Functional_Test_24 )
   END_RUNG
   RUNG wire#w1
      Contact( #In_Functional_Test.Electrical_Current_Test_Approved_PLC_Functional_Test_24 )
      Coil( #Out_Functional_Test.Electrical_Current_Test_Approved_PLC_Functional_Test_24 )
   END_RUNG
   RUNG wire#w1
      Contact( #In_Functional_Test.Visual_Test_Approved_PLC_Functional_Test_24 )
      Coil( #Out_Functional_Test.Visual_Test_Approved_PLC_Functional_Test_24 )
   END_RUNG
   RUNG wire#w1
      Move(in := #In_Functional_Test.Electrical_Current_Read_PLC_Functional_Test_24, out1 => #Out_Functional_Test.Electrical_Current_Read_PLC_Functional_Test_24)
   END_RUNG
   RUNG wire#w1
      Contact( #In_Functional_Test.Life_Trigger_PLC_Functional_Test_26 )
      Coil( #Out_Functional_Test.Life_Trigger_PLC_Functional_Test_26 )
   END_RUNG
   RUNG wire#w1
      Contact( #In_Functional_Test.Star_Test_PLC_Functional_Test_26 )
      Coil( #Out_Functional_Test.Star_Test_PLC_Functional_Test_26 )
   END_RUNG
   RUNG wire#w1
      Contact( #In_Functional_Test.Button_PLC_Functional_Test_26 )
      Coil( #Out_Functional_Test.Button_PLC_Functional_Test_26 )
   END_RUNG
   RUNG wire#w1
      Contact( #In_Functional_Test.Electrical_Current_Test_Approved_PLC_Functional_Test_26 )
      Coil( #Out_Functional_Test.Electrical_Current_Test_Approved_PLC_Functional_Test_26 )
   END_RUNG
   RUNG wire#w1
      Contact( #In_Functional_Test.Visual_Test_Approved_PLC_Functional_Test_26 )
      Coil( #Out_Functional_Test.Visual_Test_Approved_PLC_Functional_Test_26 )
   END_RUNG
   RUNG wire#w1
      Move(in := #In_Functional_Test.Electrical_Current_Read_PLC_Functional_Test_26, out1 => #Out_Functional_Test.Electrical_Current_Read_PLC_Functional_Test_26)
   END_RUNG
   RUNG wire#w1
      Contact( #In_Functional_Test.Life_Trigger_PLC_Functional_Test_28 )
      Coil( #Out_Functional_Test.Life_Trigger_PLC_Functional_Test_28 )
   END_RUNG
   RUNG wire#w1
      Contact( #In_Functional_Test.Star_Test_PLC_Functional_Test_28 )
      Coil( #Out_Functional_Test.Star_Test_PLC_Functional_Test_28 )
   END_RUNG
   RUNG wire#w1
      Contact( #In_Functional_Test.Button_PLC_Functional_Test_28 )
      Coil( #Out_Functional_Test.Button_PLC_Functional_Test_28 )
   END_RUNG
   RUNG wire#w1
      Contact( #In_Functional_Test.Electrical_Current_Test_Approved_PLC_Functional_Test_28 )
      Coil( #Out_Functional_Test.Electrical_Current_Test_Approved_PLC_Functional_Test_28 )
   END_RUNG
   RUNG wire#w1
      Contact( #In_Functional_Test.Visual_Test_Approved_PLC_Functional_Test_28 )
      Coil( #Out_Functional_Test.Visual_Test_Approved_PLC_Functional_Test_28 )
   END_RUNG
   RUNG wire#w1
      Move(in := #In_Functional_Test.Electrical_Current_Read_PLC_Functional_Test_28, out1 => #Out_Functional_Test.Electrical_Current_Read_PLC_Functional_Test_28)
   END_RUNG
   RUNG wire#w1
      Contact( #In_Functional_Test.Life_Trigger_PLC_Functional_Test_30 )
      Coil( #Out_Functional_Test.Life_Trigger_PLC_Functional_Test_30 )
   END_RUNG
   RUNG wire#w1
      Contact( #In_Functional_Test.Star_Test_PLC_Functional_Test_30 )
      Coil( #Out_Functional_Test.Star_Test_PLC_Functional_Test_30 )
   END_RUNG
   RUNG wire#w1
      Contact( #In_Functional_Test.Button_PLC_Functional_Test_30 )
      Coil( #Out_Functional_Test.Button_PLC_Functional_Test_30 )
   END_RUNG
   RUNG wire#w1
      Contact( #In_Functional_Test.Electrical_Current_Test_Approved_PLC_Functional_Test_30 )
      Coil( #Out_Functional_Test.Electrical_Current_Test_Approved_PLC_Functional_Test_30 )
   END_RUNG
   RUNG wire#w1
      Contact( #In_Functional_Test.Visual_Test_Approved_PLC_Functional_Test_30 )
      Coil( #Out_Functional_Test.Visual_Test_Approved_PLC_Functional_Test_30 )
   END_RUNG
   RUNG wire#w1
      Move(in := #In_Functional_Test.Electrical_Current_Read_PLC_Functional_Test_30, out1 => #Out_Functional_Test.Electrical_Current_Read_PLC_Functional_Test_30)
   END_RUNG
   // the same network as SCL:
   #_w1 := #Test_Station = 22;
   #Out_Functional_Test.Life_Trigger_PLC_Functional_Test_22 := #_w1 AND #Life_Trigger;
   #Out_Functional_Test.Star_Test_PLC_Functional_Test_22 := #_w1 AND #Star_Test;
   #Out_Functional_Test.Button_PLC_Functional_Test_22 := #_w1 AND #Button_Start_Approve;
   #Out_Functional_Test.Electrical_Current_Test_Approved_PLC_Functional_Test_22 := #_w1 AND #Electrical_Current_Test_Approved;
   #Out_Functional_Test.Visual_Test_Approved_PLC_Functional_Test_22 := #_w1 AND #Visual_Test_Approved;
   #Reset_Functional_Test := #_w1 AND #In_Test_Parameters.Reset_PLC_Functional_Test_22;
   IF #_w1 THEN
       #Out_Functional_Test.Electrical_Current_Read_PLC_Functional_Test_22 := #Electrical_Current_Read;
   END_IF;
   #Out_Functional_Test.Life_Trigger_PLC_Functional_Test_24 := #_w1 AND #In_Functional_Test.Life_Trigger_PLC_Functional_Test_24;
   #Out_Functional_Test.Star_Test_PLC_Functional_Test_24 := #_w1 AND #In_Functional_Test.Star_Test_PLC_Functional_Test_24;
   #Out_Functional_Test.Button_PLC_Functional_Test_24 := #_w1 AND #In_Functional_Test.Button_PLC_Functional_Test_24;
   #Out_Functional_Test.Electrical_Current_Test_Approved_PLC_Functional_Test_24 := #_w1 AND #In_Functional_Test.Electrical_Current_Test_Approved_PLC_Functional_Test_24;
   #Out_Functional_Test.Visual_Test_Approved_PLC_Functional_Test_24 := #_w1 AND #In_Functional_Test.Visual_Test_Approved_PLC_Functional_Test_24;
   IF #_w1 THEN
       #Out_Functional_Test.Electrical_Current_Read_PLC_Functional_Test_24 := #In_Functional_Test.Electrical_Current_Read_PLC_Functional_Test_24;
   END_IF;
   #Out_Functional_Test.Life_Trigger_PLC_Functional_Test_26 := #_w1 AND #In_Functional_Test.Life_Trigger_PLC_Functional_Test_26;
   #Out_Functional_Test.Star_Test_PLC_Functional_Test_26 := #_w1 AND #In_Functional_Test.Star_Test_PLC_Functional_Test_26;
   #Out_Functional_Test.Button_PLC_Functional_Test_26 := #_w1 AND #In_Functional_Test.Button_PLC_Functional_Test_26;
   #Out_Functional_Test.Electrical_Current_Test_Approved_PLC_Functional_Test_26 := #_w1 AND #In_Functional_Test.Electrical_Current_Test_Approved_PLC_Functional_Test_26;
   #Out_Functional_Test.Visual_Test_Approved_PLC_Functional_Test_26 := #_w1 AND #In_Functional_Test.Visual_Test_Approved_PLC_Functional_Test_26;
   IF #_w1 THEN
       #Out_Functional_Test.Electrical_Current_Read_PLC_Functional_Test_26 := #In_Functional_Test.Electrical_Current_Read_PLC_Functional_Test_26;
   END_IF;
   #Out_Functional_Test.Life_Trigger_PLC_Functional_Test_28 := #_w1 AND #In_Functional_Test.Life_Trigger_PLC_Functional_Test_28;
   #Out_Functional_Test.Star_Test_PLC_Functional_Test_28 := #_w1 AND #In_Functional_Test.Star_Test_PLC_Functional_Test_28;
   #Out_Functional_Test.Button_PLC_Functional_Test_28 := #_w1 AND #In_Functional_Test.Button_PLC_Functional_Test_28;
   #Out_Functional_Test.Electrical_Current_Test_Approved_PLC_Functional_Test_28 := #_w1 AND #In_Functional_Test.Electrical_Current_Test_Approved_PLC_Functional_Test_28;
   #Out_Functional_Test.Visual_Test_Approved_PLC_Functional_Test_28 := #_w1 AND #In_Functional_Test.Visual_Test_Approved_PLC_Functional_Test_28;
   IF #_w1 THEN
       #Out_Functional_Test.Electrical_Current_Read_PLC_Functional_Test_28 := #In_Functional_Test.Electrical_Current_Read_PLC_Functional_Test_28;
   END_IF;
   #Out_Functional_Test.Life_Trigger_PLC_Functional_Test_30 := #_w1 AND #In_Functional_Test.Life_Trigger_PLC_Functional_Test_30;
   #Out_Functional_Test.Star_Test_PLC_Functional_Test_30 := #_w1 AND #In_Functional_Test.Star_Test_PLC_Functional_Test_30;
   #Out_Functional_Test.Button_PLC_Functional_Test_30 := #_w1 AND #In_Functional_Test.Button_PLC_Functional_Test_30;
   #Out_Functional_Test.Electrical_Current_Test_Approved_PLC_Functional_Test_30 := #_w1 AND #In_Functional_Test.Electrical_Current_Test_Approved_PLC_Functional_Test_30;
   #Out_Functional_Test.Visual_Test_Approved_PLC_Functional_Test_30 := #_w1 AND #In_Functional_Test.Visual_Test_Approved_PLC_Functional_Test_30;
   IF #_w1 THEN
       #Out_Functional_Test.Electrical_Current_Read_PLC_Functional_Test_30 := #In_Functional_Test.Electrical_Current_Read_PLC_Functional_Test_30;
   END_IF;
END_REGION

REGION Network 13: Functional Test Station 24
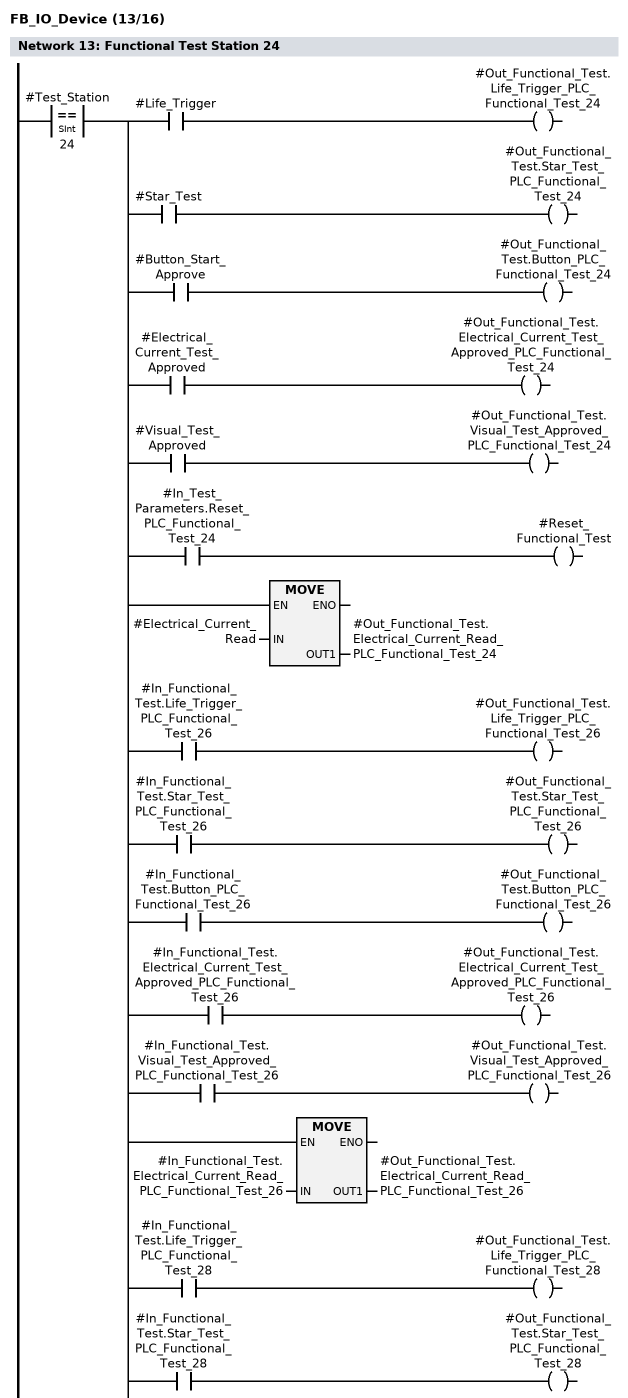
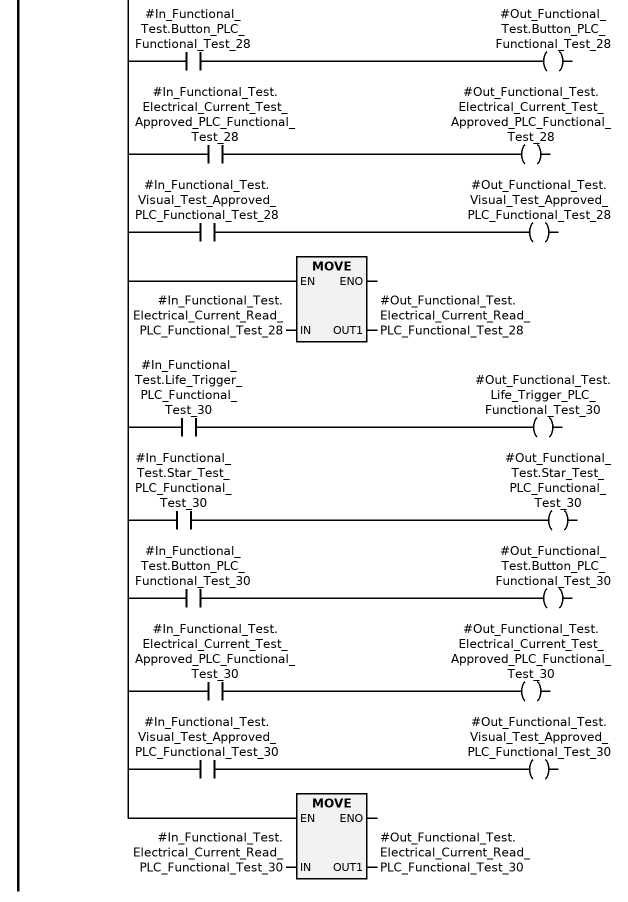
   RUNG wire#powerrail
      { S7_Templates := "SrcType := SInt" } EQ_Contact(in1 := #Test_Station, in2 := 24)
      wire#w1
      Contact( #Life_Trigger )
      Coil( #Out_Functional_Test.Life_Trigger_PLC_Functional_Test_24 )
   END_RUNG
   RUNG wire#w1
      Contact( #Star_Test )
      Coil( #Out_Functional_Test.Star_Test_PLC_Functional_Test_24 )
   END_RUNG
   RUNG wire#w1
      Contact( #Button_Start_Approve )
      Coil( #Out_Functional_Test.Button_PLC_Functional_Test_24 )
   END_RUNG
   RUNG wire#w1
      Contact( #Electrical_Current_Test_Approved )
      Coil( #Out_Functional_Test.Electrical_Current_Test_Approved_PLC_Functional_Test_24 )
   END_RUNG
   RUNG wire#w1
      Contact( #Visual_Test_Approved )
      Coil( #Out_Functional_Test.Visual_Test_Approved_PLC_Functional_Test_24 )
   END_RUNG
   RUNG wire#w1
      Contact( #In_Test_Parameters.Reset_PLC_Functional_Test_24 )
      Coil( #Reset_Functional_Test )
   END_RUNG
   RUNG wire#w1
      Move(in := #Electrical_Current_Read, out1 => #Out_Functional_Test.Electrical_Current_Read_PLC_Functional_Test_24)
   END_RUNG
   RUNG wire#w1
      Contact( #In_Functional_Test.Life_Trigger_PLC_Functional_Test_26 )
      Coil( #Out_Functional_Test.Life_Trigger_PLC_Functional_Test_26 )
   END_RUNG
   RUNG wire#w1
      Contact( #In_Functional_Test.Star_Test_PLC_Functional_Test_26 )
      Coil( #Out_Functional_Test.Star_Test_PLC_Functional_Test_26 )
   END_RUNG
   RUNG wire#w1
      Contact( #In_Functional_Test.Button_PLC_Functional_Test_26 )
      Coil( #Out_Functional_Test.Button_PLC_Functional_Test_26 )
   END_RUNG
   RUNG wire#w1
      Contact( #In_Functional_Test.Electrical_Current_Test_Approved_PLC_Functional_Test_26 )
      Coil( #Out_Functional_Test.Electrical_Current_Test_Approved_PLC_Functional_Test_26 )
   END_RUNG
   RUNG wire#w1
      Contact( #In_Functional_Test.Visual_Test_Approved_PLC_Functional_Test_26 )
      Coil( #Out_Functional_Test.Visual_Test_Approved_PLC_Functional_Test_26 )
   END_RUNG
   RUNG wire#w1
      Move(in := #In_Functional_Test.Electrical_Current_Read_PLC_Functional_Test_26, out1 => #Out_Functional_Test.Electrical_Current_Read_PLC_Functional_Test_26)
   END_RUNG
   RUNG wire#w1
      Contact( #In_Functional_Test.Life_Trigger_PLC_Functional_Test_28 )
      Coil( #Out_Functional_Test.Life_Trigger_PLC_Functional_Test_28 )
   END_RUNG
   RUNG wire#w1
      Contact( #In_Functional_Test.Star_Test_PLC_Functional_Test_28 )
      Coil( #Out_Functional_Test.Star_Test_PLC_Functional_Test_28 )
   END_RUNG
   RUNG wire#w1
      Contact( #In_Functional_Test.Button_PLC_Functional_Test_28 )
      Coil( #Out_Functional_Test.Button_PLC_Functional_Test_28 )
   END_RUNG
   RUNG wire#w1
      Contact( #In_Functional_Test.Electrical_Current_Test_Approved_PLC_Functional_Test_28 )
      Coil( #Out_Functional_Test.Electrical_Current_Test_Approved_PLC_Functional_Test_28 )
   END_RUNG
   RUNG wire#w1
      Contact( #In_Functional_Test.Visual_Test_Approved_PLC_Functional_Test_28 )
      Coil( #Out_Functional_Test.Visual_Test_Approved_PLC_Functional_Test_28 )
   END_RUNG
   RUNG wire#w1
      Move(in := #In_Functional_Test.Electrical_Current_Read_PLC_Functional_Test_28, out1 => #Out_Functional_Test.Electrical_Current_Read_PLC_Functional_Test_28)
   END_RUNG
   RUNG wire#w1
      Contact( #In_Functional_Test.Life_Trigger_PLC_Functional_Test_30 )
      Coil( #Out_Functional_Test.Life_Trigger_PLC_Functional_Test_30 )
   END_RUNG
   RUNG wire#w1
      Contact( #In_Functional_Test.Star_Test_PLC_Functional_Test_30 )
      Coil( #Out_Functional_Test.Star_Test_PLC_Functional_Test_30 )
   END_RUNG
   RUNG wire#w1
      Contact( #In_Functional_Test.Button_PLC_Functional_Test_30 )
      Coil( #Out_Functional_Test.Button_PLC_Functional_Test_30 )
   END_RUNG
   RUNG wire#w1
      Contact( #In_Functional_Test.Electrical_Current_Test_Approved_PLC_Functional_Test_30 )
      Coil( #Out_Functional_Test.Electrical_Current_Test_Approved_PLC_Functional_Test_30 )
   END_RUNG
   RUNG wire#w1
      Contact( #In_Functional_Test.Visual_Test_Approved_PLC_Functional_Test_30 )
      Coil( #Out_Functional_Test.Visual_Test_Approved_PLC_Functional_Test_30 )
   END_RUNG
   RUNG wire#w1
      Move(in := #In_Functional_Test.Electrical_Current_Read_PLC_Functional_Test_30, out1 => #Out_Functional_Test.Electrical_Current_Read_PLC_Functional_Test_30)
   END_RUNG
   // the same network as SCL:
   #_w1 := #Test_Station = 24;
   #Out_Functional_Test.Life_Trigger_PLC_Functional_Test_24 := #_w1 AND #Life_Trigger;
   #Out_Functional_Test.Star_Test_PLC_Functional_Test_24 := #_w1 AND #Star_Test;
   #Out_Functional_Test.Button_PLC_Functional_Test_24 := #_w1 AND #Button_Start_Approve;
   #Out_Functional_Test.Electrical_Current_Test_Approved_PLC_Functional_Test_24 := #_w1 AND #Electrical_Current_Test_Approved;
   #Out_Functional_Test.Visual_Test_Approved_PLC_Functional_Test_24 := #_w1 AND #Visual_Test_Approved;
   #Reset_Functional_Test := #_w1 AND #In_Test_Parameters.Reset_PLC_Functional_Test_24;
   IF #_w1 THEN
       #Out_Functional_Test.Electrical_Current_Read_PLC_Functional_Test_24 := #Electrical_Current_Read;
   END_IF;
   #Out_Functional_Test.Life_Trigger_PLC_Functional_Test_26 := #_w1 AND #In_Functional_Test.Life_Trigger_PLC_Functional_Test_26;
   #Out_Functional_Test.Star_Test_PLC_Functional_Test_26 := #_w1 AND #In_Functional_Test.Star_Test_PLC_Functional_Test_26;
   #Out_Functional_Test.Button_PLC_Functional_Test_26 := #_w1 AND #In_Functional_Test.Button_PLC_Functional_Test_26;
   #Out_Functional_Test.Electrical_Current_Test_Approved_PLC_Functional_Test_26 := #_w1 AND #In_Functional_Test.Electrical_Current_Test_Approved_PLC_Functional_Test_26;
   #Out_Functional_Test.Visual_Test_Approved_PLC_Functional_Test_26 := #_w1 AND #In_Functional_Test.Visual_Test_Approved_PLC_Functional_Test_26;
   IF #_w1 THEN
       #Out_Functional_Test.Electrical_Current_Read_PLC_Functional_Test_26 := #In_Functional_Test.Electrical_Current_Read_PLC_Functional_Test_26;
   END_IF;
   #Out_Functional_Test.Life_Trigger_PLC_Functional_Test_28 := #_w1 AND #In_Functional_Test.Life_Trigger_PLC_Functional_Test_28;
   #Out_Functional_Test.Star_Test_PLC_Functional_Test_28 := #_w1 AND #In_Functional_Test.Star_Test_PLC_Functional_Test_28;
   #Out_Functional_Test.Button_PLC_Functional_Test_28 := #_w1 AND #In_Functional_Test.Button_PLC_Functional_Test_28;
   #Out_Functional_Test.Electrical_Current_Test_Approved_PLC_Functional_Test_28 := #_w1 AND #In_Functional_Test.Electrical_Current_Test_Approved_PLC_Functional_Test_28;
   #Out_Functional_Test.Visual_Test_Approved_PLC_Functional_Test_28 := #_w1 AND #In_Functional_Test.Visual_Test_Approved_PLC_Functional_Test_28;
   IF #_w1 THEN
       #Out_Functional_Test.Electrical_Current_Read_PLC_Functional_Test_28 := #In_Functional_Test.Electrical_Current_Read_PLC_Functional_Test_28;
   END_IF;
   #Out_Functional_Test.Life_Trigger_PLC_Functional_Test_30 := #_w1 AND #In_Functional_Test.Life_Trigger_PLC_Functional_Test_30;
   #Out_Functional_Test.Star_Test_PLC_Functional_Test_30 := #_w1 AND #In_Functional_Test.Star_Test_PLC_Functional_Test_30;
   #Out_Functional_Test.Button_PLC_Functional_Test_30 := #_w1 AND #In_Functional_Test.Button_PLC_Functional_Test_30;
   #Out_Functional_Test.Electrical_Current_Test_Approved_PLC_Functional_Test_30 := #_w1 AND #In_Functional_Test.Electrical_Current_Test_Approved_PLC_Functional_Test_30;
   #Out_Functional_Test.Visual_Test_Approved_PLC_Functional_Test_30 := #_w1 AND #In_Functional_Test.Visual_Test_Approved_PLC_Functional_Test_30;
   IF #_w1 THEN
       #Out_Functional_Test.Electrical_Current_Read_PLC_Functional_Test_30 := #In_Functional_Test.Electrical_Current_Read_PLC_Functional_Test_30;
   END_IF;
END_REGION

REGION Network 14: Functional Test Station 26
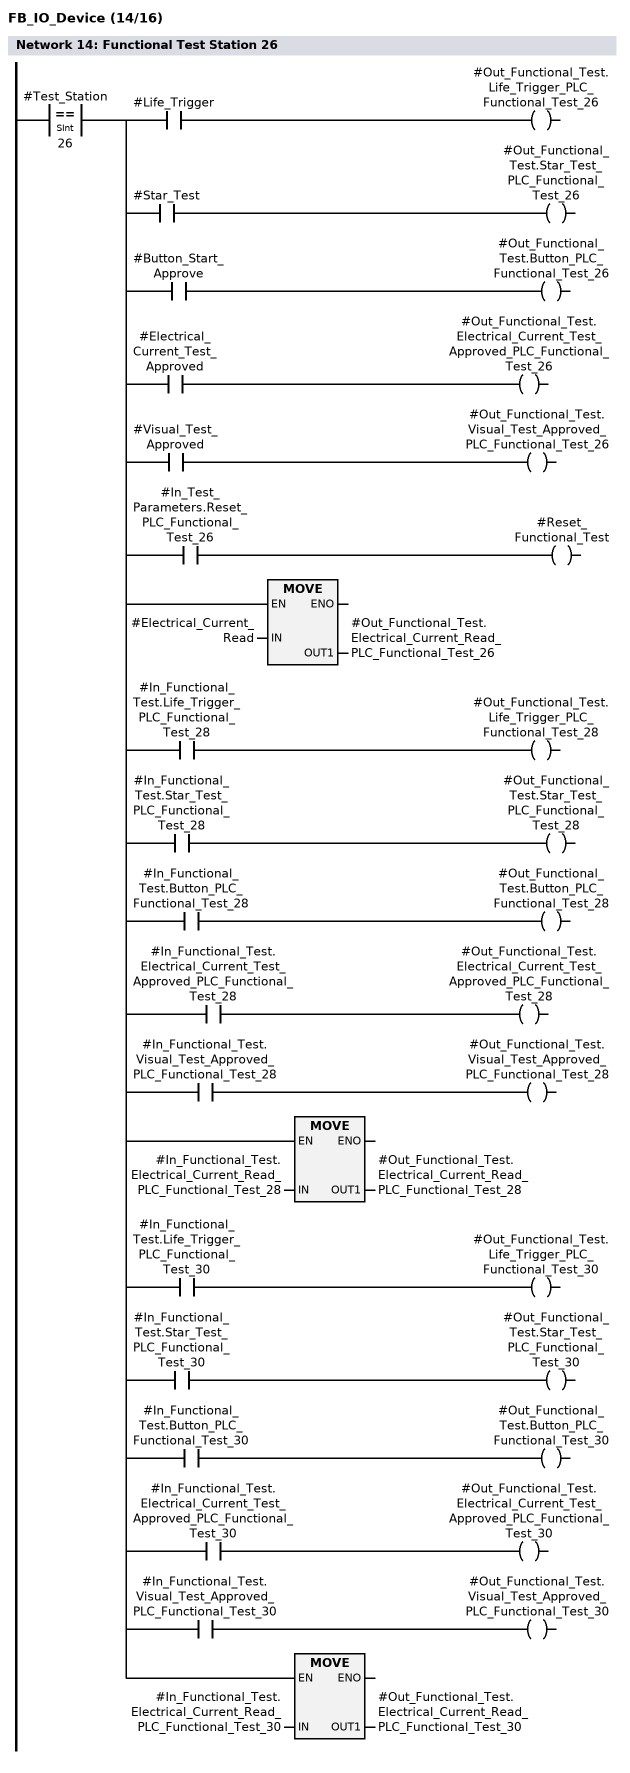
   RUNG wire#powerrail
      { S7_Templates := "SrcType := SInt" } EQ_Contact(in1 := #Test_Station, in2 := 26)
      wire#w1
      Contact( #Life_Trigger )
      Coil( #Out_Functional_Test.Life_Trigger_PLC_Functional_Test_26 )
   END_RUNG
   RUNG wire#w1
      Contact( #Star_Test )
      Coil( #Out_Functional_Test.Star_Test_PLC_Functional_Test_26 )
   END_RUNG
   RUNG wire#w1
      Contact( #Button_Start_Approve )
      Coil( #Out_Functional_Test.Button_PLC_Functional_Test_26 )
   END_RUNG
   RUNG wire#w1
      Contact( #Electrical_Current_Test_Approved )
      Coil( #Out_Functional_Test.Electrical_Current_Test_Approved_PLC_Functional_Test_26 )
   END_RUNG
   RUNG wire#w1
      Contact( #Visual_Test_Approved )
      Coil( #Out_Functional_Test.Visual_Test_Approved_PLC_Functional_Test_26 )
   END_RUNG
   RUNG wire#w1
      Contact( #In_Test_Parameters.Reset_PLC_Functional_Test_26 )
      Coil( #Reset_Functional_Test )
   END_RUNG
   RUNG wire#w1
      Move(in := #Electrical_Current_Read, out1 => #Out_Functional_Test.Electrical_Current_Read_PLC_Functional_Test_26)
   END_RUNG
   RUNG wire#w1
      Contact( #In_Functional_Test.Life_Trigger_PLC_Functional_Test_28 )
      Coil( #Out_Functional_Test.Life_Trigger_PLC_Functional_Test_28 )
   END_RUNG
   RUNG wire#w1
      Contact( #In_Functional_Test.Star_Test_PLC_Functional_Test_28 )
      Coil( #Out_Functional_Test.Star_Test_PLC_Functional_Test_28 )
   END_RUNG
   RUNG wire#w1
      Contact( #In_Functional_Test.Button_PLC_Functional_Test_28 )
      Coil( #Out_Functional_Test.Button_PLC_Functional_Test_28 )
   END_RUNG
   RUNG wire#w1
      Contact( #In_Functional_Test.Electrical_Current_Test_Approved_PLC_Functional_Test_28 )
      Coil( #Out_Functional_Test.Electrical_Current_Test_Approved_PLC_Functional_Test_28 )
   END_RUNG
   RUNG wire#w1
      Contact( #In_Functional_Test.Visual_Test_Approved_PLC_Functional_Test_28 )
      Coil( #Out_Functional_Test.Visual_Test_Approved_PLC_Functional_Test_28 )
   END_RUNG
   RUNG wire#w1
      Move(in := #In_Functional_Test.Electrical_Current_Read_PLC_Functional_Test_28, out1 => #Out_Functional_Test.Electrical_Current_Read_PLC_Functional_Test_28)
   END_RUNG
   RUNG wire#w1
      Contact( #In_Functional_Test.Life_Trigger_PLC_Functional_Test_30 )
      Coil( #Out_Functional_Test.Life_Trigger_PLC_Functional_Test_30 )
   END_RUNG
   RUNG wire#w1
      Contact( #In_Functional_Test.Star_Test_PLC_Functional_Test_30 )
      Coil( #Out_Functional_Test.Star_Test_PLC_Functional_Test_30 )
   END_RUNG
   RUNG wire#w1
      Contact( #In_Functional_Test.Button_PLC_Functional_Test_30 )
      Coil( #Out_Functional_Test.Button_PLC_Functional_Test_30 )
   END_RUNG
   RUNG wire#w1
      Contact( #In_Functional_Test.Electrical_Current_Test_Approved_PLC_Functional_Test_30 )
      Coil( #Out_Functional_Test.Electrical_Current_Test_Approved_PLC_Functional_Test_30 )
   END_RUNG
   RUNG wire#w1
      Contact( #In_Functional_Test.Visual_Test_Approved_PLC_Functional_Test_30 )
      Coil( #Out_Functional_Test.Visual_Test_Approved_PLC_Functional_Test_30 )
   END_RUNG
   RUNG wire#w1
      Move(in := #In_Functional_Test.Electrical_Current_Read_PLC_Functional_Test_30, out1 => #Out_Functional_Test.Electrical_Current_Read_PLC_Functional_Test_30)
   END_RUNG
   // the same network as SCL:
   #_w1 := #Test_Station = 26;
   #Out_Functional_Test.Life_Trigger_PLC_Functional_Test_26 := #_w1 AND #Life_Trigger;
   #Out_Functional_Test.Star_Test_PLC_Functional_Test_26 := #_w1 AND #Star_Test;
   #Out_Functional_Test.Button_PLC_Functional_Test_26 := #_w1 AND #Button_Start_Approve;
   #Out_Functional_Test.Electrical_Current_Test_Approved_PLC_Functional_Test_26 := #_w1 AND #Electrical_Current_Test_Approved;
   #Out_Functional_Test.Visual_Test_Approved_PLC_Functional_Test_26 := #_w1 AND #Visual_Test_Approved;
   #Reset_Functional_Test := #_w1 AND #In_Test_Parameters.Reset_PLC_Functional_Test_26;
   IF #_w1 THEN
       #Out_Functional_Test.Electrical_Current_Read_PLC_Functional_Test_26 := #Electrical_Current_Read;
   END_IF;
   #Out_Functional_Test.Life_Trigger_PLC_Functional_Test_28 := #_w1 AND #In_Functional_Test.Life_Trigger_PLC_Functional_Test_28;
   #Out_Functional_Test.Star_Test_PLC_Functional_Test_28 := #_w1 AND #In_Functional_Test.Star_Test_PLC_Functional_Test_28;
   #Out_Functional_Test.Button_PLC_Functional_Test_28 := #_w1 AND #In_Functional_Test.Button_PLC_Functional_Test_28;
   #Out_Functional_Test.Electrical_Current_Test_Approved_PLC_Functional_Test_28 := #_w1 AND #In_Functional_Test.Electrical_Current_Test_Approved_PLC_Functional_Test_28;
   #Out_Functional_Test.Visual_Test_Approved_PLC_Functional_Test_28 := #_w1 AND #In_Functional_Test.Visual_Test_Approved_PLC_Functional_Test_28;
   IF #_w1 THEN
       #Out_Functional_Test.Electrical_Current_Read_PLC_Functional_Test_28 := #In_Functional_Test.Electrical_Current_Read_PLC_Functional_Test_28;
   END_IF;
   #Out_Functional_Test.Life_Trigger_PLC_Functional_Test_30 := #_w1 AND #In_Functional_Test.Life_Trigger_PLC_Functional_Test_30;
   #Out_Functional_Test.Star_Test_PLC_Functional_Test_30 := #_w1 AND #In_Functional_Test.Star_Test_PLC_Functional_Test_30;
   #Out_Functional_Test.Button_PLC_Functional_Test_30 := #_w1 AND #In_Functional_Test.Button_PLC_Functional_Test_30;
   #Out_Functional_Test.Electrical_Current_Test_Approved_PLC_Functional_Test_30 := #_w1 AND #In_Functional_Test.Electrical_Current_Test_Approved_PLC_Functional_Test_30;
   #Out_Functional_Test.Visual_Test_Approved_PLC_Functional_Test_30 := #_w1 AND #In_Functional_Test.Visual_Test_Approved_PLC_Functional_Test_30;
   IF #_w1 THEN
       #Out_Functional_Test.Electrical_Current_Read_PLC_Functional_Test_30 := #In_Functional_Test.Electrical_Current_Read_PLC_Functional_Test_30;
   END_IF;
END_REGION

REGION Network 15: Functional Test Station 28
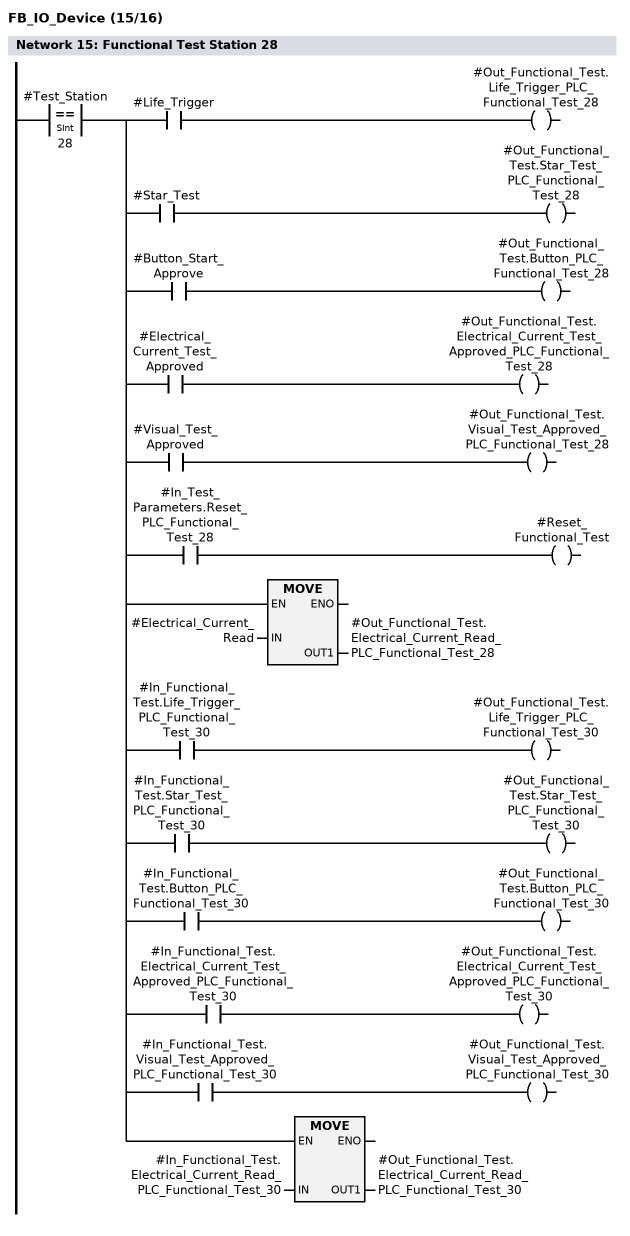
   RUNG wire#powerrail
      { S7_Templates := "SrcType := SInt" } EQ_Contact(in1 := #Test_Station, in2 := 28)
      wire#w1
      Contact( #Life_Trigger )
      Coil( #Out_Functional_Test.Life_Trigger_PLC_Functional_Test_28 )
   END_RUNG
   RUNG wire#w1
      Contact( #Star_Test )
      Coil( #Out_Functional_Test.Star_Test_PLC_Functional_Test_28 )
   END_RUNG
   RUNG wire#w1
      Contact( #Button_Start_Approve )
      Coil( #Out_Functional_Test.Button_PLC_Functional_Test_28 )
   END_RUNG
   RUNG wire#w1
      Contact( #Electrical_Current_Test_Approved )
      Coil( #Out_Functional_Test.Electrical_Current_Test_Approved_PLC_Functional_Test_28 )
   END_RUNG
   RUNG wire#w1
      Contact( #Visual_Test_Approved )
      Coil( #Out_Functional_Test.Visual_Test_Approved_PLC_Functional_Test_28 )
   END_RUNG
   RUNG wire#w1
      Contact( #In_Test_Parameters.Reset_PLC_Functional_Test_28 )
      Coil( #Reset_Functional_Test )
   END_RUNG
   RUNG wire#w1
      Move(in := #Electrical_Current_Read, out1 => #Out_Functional_Test.Electrical_Current_Read_PLC_Functional_Test_28)
   END_RUNG
   RUNG wire#w1
      Contact( #In_Functional_Test.Life_Trigger_PLC_Functional_Test_30 )
      Coil( #Out_Functional_Test.Life_Trigger_PLC_Functional_Test_30 )
   END_RUNG
   RUNG wire#w1
      Contact( #In_Functional_Test.Star_Test_PLC_Functional_Test_30 )
      Coil( #Out_Functional_Test.Star_Test_PLC_Functional_Test_30 )
   END_RUNG
   RUNG wire#w1
      Contact( #In_Functional_Test.Button_PLC_Functional_Test_30 )
      Coil( #Out_Functional_Test.Button_PLC_Functional_Test_30 )
   END_RUNG
   RUNG wire#w1
      Contact( #In_Functional_Test.Electrical_Current_Test_Approved_PLC_Functional_Test_30 )
      Coil( #Out_Functional_Test.Electrical_Current_Test_Approved_PLC_Functional_Test_30 )
   END_RUNG
   RUNG wire#w1
      Contact( #In_Functional_Test.Visual_Test_Approved_PLC_Functional_Test_30 )
      Coil( #Out_Functional_Test.Visual_Test_Approved_PLC_Functional_Test_30 )
   END_RUNG
   RUNG wire#w1
      Move(in := #In_Functional_Test.Electrical_Current_Read_PLC_Functional_Test_30, out1 => #Out_Functional_Test.Electrical_Current_Read_PLC_Functional_Test_30)
   END_RUNG
   // the same network as SCL:
   #_w1 := #Test_Station = 28;
   #Out_Functional_Test.Life_Trigger_PLC_Functional_Test_28 := #_w1 AND #Life_Trigger;
   #Out_Functional_Test.Star_Test_PLC_Functional_Test_28 := #_w1 AND #Star_Test;
   #Out_Functional_Test.Button_PLC_Functional_Test_28 := #_w1 AND #Button_Start_Approve;
   #Out_Functional_Test.Electrical_Current_Test_Approved_PLC_Functional_Test_28 := #_w1 AND #Electrical_Current_Test_Approved;
   #Out_Functional_Test.Visual_Test_Approved_PLC_Functional_Test_28 := #_w1 AND #Visual_Test_Approved;
   #Reset_Functional_Test := #_w1 AND #In_Test_Parameters.Reset_PLC_Functional_Test_28;
   IF #_w1 THEN
       #Out_Functional_Test.Electrical_Current_Read_PLC_Functional_Test_28 := #Electrical_Current_Read;
   END_IF;
   #Out_Functional_Test.Life_Trigger_PLC_Functional_Test_30 := #_w1 AND #In_Functional_Test.Life_Trigger_PLC_Functional_Test_30;
   #Out_Functional_Test.Star_Test_PLC_Functional_Test_30 := #_w1 AND #In_Functional_Test.Star_Test_PLC_Functional_Test_30;
   #Out_Functional_Test.Button_PLC_Functional_Test_30 := #_w1 AND #In_Functional_Test.Button_PLC_Functional_Test_30;
   #Out_Functional_Test.Electrical_Current_Test_Approved_PLC_Functional_Test_30 := #_w1 AND #In_Functional_Test.Electrical_Current_Test_Approved_PLC_Functional_Test_30;
   #Out_Functional_Test.Visual_Test_Approved_PLC_Functional_Test_30 := #_w1 AND #In_Functional_Test.Visual_Test_Approved_PLC_Functional_Test_30;
   IF #_w1 THEN
       #Out_Functional_Test.Electrical_Current_Read_PLC_Functional_Test_30 := #In_Functional_Test.Electrical_Current_Read_PLC_Functional_Test_30;
   END_IF;
END_REGION

REGION Network 16: Functional Test Station 30
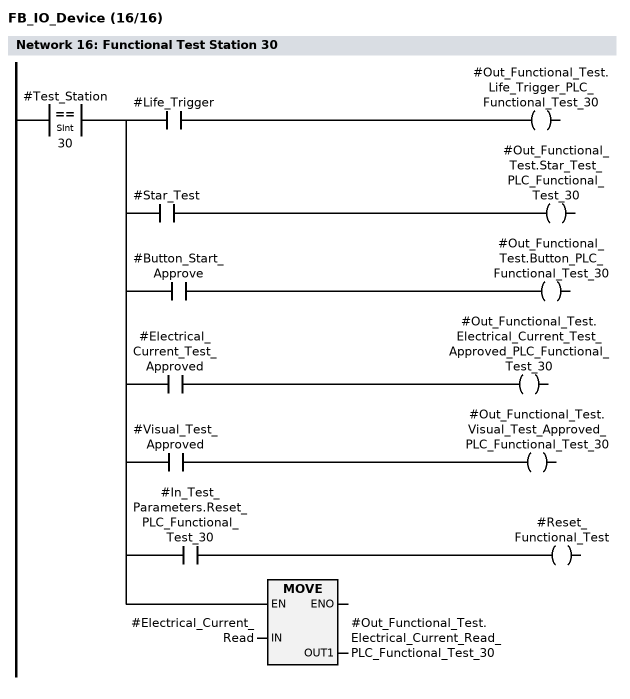
   RUNG wire#powerrail
      { S7_Templates := "SrcType := SInt" } EQ_Contact(in1 := #Test_Station, in2 := 30)
      wire#w1
      Contact( #Life_Trigger )
      Coil( #Out_Functional_Test.Life_Trigger_PLC_Functional_Test_30 )
   END_RUNG
   RUNG wire#w1
      Contact( #Star_Test )
      Coil( #Out_Functional_Test.Star_Test_PLC_Functional_Test_30 )
   END_RUNG
   RUNG wire#w1
      Contact( #Button_Start_Approve )
      Coil( #Out_Functional_Test.Button_PLC_Functional_Test_30 )
   END_RUNG
   RUNG wire#w1
      Contact( #Electrical_Current_Test_Approved )
      Coil( #Out_Functional_Test.Electrical_Current_Test_Approved_PLC_Functional_Test_30 )
   END_RUNG
   RUNG wire#w1
      Contact( #Visual_Test_Approved )
      Coil( #Out_Functional_Test.Visual_Test_Approved_PLC_Functional_Test_30 )
   END_RUNG
   RUNG wire#w1
      Contact( #In_Test_Parameters.Reset_PLC_Functional_Test_30 )
      Coil( #Reset_Functional_Test )
   END_RUNG
   RUNG wire#w1
      Move(in := #Electrical_Current_Read, out1 => #Out_Functional_Test.Electrical_Current_Read_PLC_Functional_Test_30)
   END_RUNG
   // the same network as SCL:
   #_w1 := #Test_Station = 30;
   #Out_Functional_Test.Life_Trigger_PLC_Functional_Test_30 := #_w1 AND #Life_Trigger;
   #Out_Functional_Test.Star_Test_PLC_Functional_Test_30 := #_w1 AND #Star_Test;
   #Out_Functional_Test.Button_PLC_Functional_Test_30 := #_w1 AND #Button_Start_Approve;
   #Out_Functional_Test.Electrical_Current_Test_Approved_PLC_Functional_Test_30 := #_w1 AND #Electrical_Current_Test_Approved;
   #Out_Functional_Test.Visual_Test_Approved_PLC_Functional_Test_30 := #_w1 AND #Visual_Test_Approved;
   #Reset_Functional_Test := #_w1 AND #In_Test_Parameters.Reset_PLC_Functional_Test_30;
   IF #_w1 THEN
       #Out_Functional_Test.Electrical_Current_Read_PLC_Functional_Test_30 := #Electrical_Current_Read;
   END_IF;
END_REGION
END_FUNCTION_BLOCK

FUNCTION_BLOCK "FB_Electrical_Current_Test"   // FB6, LAD
{ S7_Optimized_Access := 'TRUE' }
// stored: MemoryReserve 100, SetENOAutomatically false
   VAR_INPUT
      Star_Functional_Test : Bool;
      Reset_Functional_Test : Bool;
      Electrical_Current_Read_UInt : UInt;
      In_Test_Parameters : "IO_Device_Test_Parameters";
   END_VAR
   VAR_OUTPUT
      Electrical_Current_Test_Approved : Bool;
   END_VAR
   VAR
      Timer_Delay_Read_Current { S7_SetPoint := 'True'} : TON_TIME;
      Timer_Delay_Reset { S7_SetPoint := 'True'} : TON_TIME;
   END_VAR
BEGIN

REGION Network 1
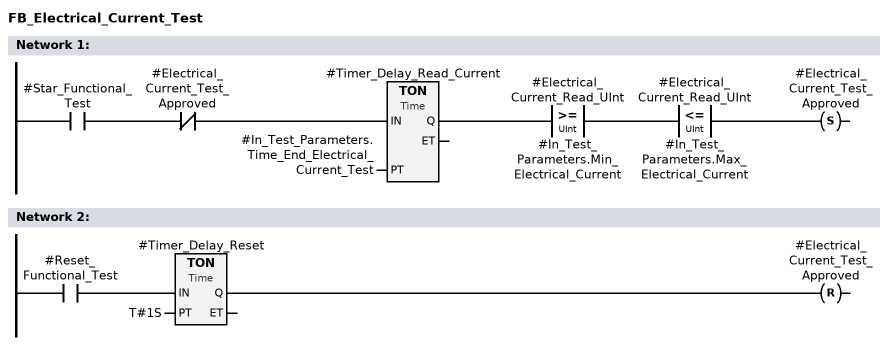
   RUNG wire#powerrail
      Contact( #Star_Functional_Test )
      I_Contact( #Electrical_Current_Test_Approved )
      { S7_Templates := "time_type := Time" } #Timer_Delay_Read_Current.TON(pt := #In_Test_Parameters.Time_End_Electrical_Current_Test, et =>)
      { S7_Templates := "SrcType := UInt" } GE_Contact(in1 := #Electrical_Current_Read_UInt, in2 := #In_Test_Parameters.Min_Electrical_Current)
      { S7_Templates := "SrcType := UInt" } LE_Contact(in1 := #Electrical_Current_Read_UInt, in2 := #In_Test_Parameters.Max_Electrical_Current)
      S_Coil( #Electrical_Current_Test_Approved )
   END_RUNG
   // the same network as SCL:
   #Timer_Delay_Read_Current(IN := #Star_Functional_Test AND NOT #Electrical_Current_Test_Approved,   // TON
                           PT := #In_Test_Parameters.Time_End_Electrical_Current_Test);
   IF #Timer_Delay_Read_Current.Q AND (#Electrical_Current_Read_UInt >= #In_Test_Parameters.Min_Electrical_Current) AND (#Electrical_Current_Read_UInt <= #In_Test_Parameters.Max_Electrical_Current) THEN
       #Electrical_Current_Test_Approved := TRUE;
   END_IF;
END_REGION

REGION Network 2
   RUNG wire#powerrail
      Contact( #Reset_Functional_Test )
      { S7_Templates := "time_type := Time" } #Timer_Delay_Reset.TON(pt := T#1S, et =>)
      R_Coil( #Electrical_Current_Test_Approved )
   END_RUNG
   // the same network as SCL:
   #Timer_Delay_Reset(IN := #Reset_Functional_Test, PT := T#1S);   // TON
   IF #Timer_Delay_Reset.Q THEN #Electrical_Current_Test_Approved := FALSE; END_IF;
END_REGION
END_FUNCTION_BLOCK

DATA_BLOCK "Instance_FB_Analogic_Input_DB"   // DB102
// stored: AutoNumber false, InstanceOfName FB_Analogic_Input, InstanceOfType FB
"FB_Analogic_Input"
   // VAR_INPUT
   //    Analogic_Input_0 { ExternalAccessible := 'False'; ExternalVisible := 'False'; ExternalWritable := 'False'} : Int;
   //    Analogic_Input_1 { ExternalAccessible := 'False'; ExternalVisible := 'False'; ExternalWritable := 'False'} : Int;
   //    Min_NormX_AI_0 { ExternalAccessible := 'False'; ExternalVisible := 'False'; ExternalWritable := 'False'} : Int;
   //    Max_NormX_AI_0 { ExternalAccessible := 'False'; ExternalVisible := 'False'; ExternalWritable := 'False'} : Int;
   //    Min_NormX_AI_1 { ExternalAccessible := 'False'; ExternalVisible := 'False'; ExternalWritable := 'False'} : Int;
   //    Max_NormX_AI_1 { ExternalAccessible := 'False'; ExternalVisible := 'False'; ExternalWritable := 'False'} : Int;
   //    Scale_Min_AI_0 { ExternalAccessible := 'False'; ExternalVisible := 'False'; ExternalWritable := 'False'} : Real;
   //    Scale_Max_AI_0 { ExternalAccessible := 'False'; ExternalVisible := 'False'; ExternalWritable := 'False'} : Real;
   //    Scale_Min_AI_1 { ExternalAccessible := 'False'; ExternalVisible := 'False'; ExternalWritable := 'False'} : Real;
   //    Scale_Max_AI_1 { ExternalAccessible := 'False'; ExternalVisible := 'False'; ExternalWritable := 'False'} : Real;
   // END_VAR
   // VAR_OUTPUT
   //    Value_Real_AI_0 { ExternalAccessible := 'False'; ExternalVisible := 'False'; ExternalWritable := 'False'} : Real;
   //    Value_Real_AI_1 { ExternalAccessible := 'False'; ExternalVisible := 'False'; ExternalWritable := 'False'} : Real;
   //    Value_UInt_AI_0 : UInt;
   //    Value_UInt_AI_1 : UInt;
   // END_VAR
   // VAR
   //    Norm_X_Out_AI_0 { ExternalAccessible := 'False'; ExternalVisible := 'False'; ExternalWritable := 'False'} : Real;
   //    Norm_X_Out_AI_1 { ExternalAccessible := 'False'; ExternalVisible := 'False'; ExternalWritable := 'False'} : Real;
   // END_VAR
BEGIN
END_DATA_BLOCK

DATA_BLOCK "Instance_FB_Digital_Outputs_DB"   // DB103
// stored: AutoNumber false, InstanceOfName FB_Digital_Outputs, InstanceOfType FB
"FB_Digital_Outputs"
BEGIN
END_DATA_BLOCK

DATA_BLOCK "Instance_FB_IO_Device_DB"   // DB104
// stored: AutoNumber false, InstanceOfName FB_IO_Device, InstanceOfType FB
"FB_IO_Device"
BEGIN
END_DATA_BLOCK

DATA_BLOCK "Instance_FB_Start_Test_DB"   // DB105
// stored: AutoNumber false, InstanceOfName FB_Start_Test, InstanceOfType FB
"FB_Start_Test"
   // VAR_INPUT
   //    Button_Start_Approve : Bool;
   //    Electrical_Current_Test_Approved : Bool;
   //    Visual_Test_Approved_PLC : Bool;
   //    Reset_Funcional_Test : Bool;
   // END_VAR
   // VAR_OUTPUT
   //    Start_Functional_Test : Bool;
   //    Blink_Button_Light : Bool;
   //    Turn_On_Button_Light : Bool;
   //    Light_Fail_Test : Bool;
   //    Light_Approve_Test : Bool;
   // END_VAR
   // VAR
   //    Aux_Trigger_0 : Bool;
   // END_VAR
BEGIN
END_DATA_BLOCK
